# B&R Automation Studio project NAEUL004C00R13L518F00 (part 32)

### Startup.typ - Do Not Change!!!
```iecst
(*2019-04-04*)
(**)

TYPE
	eStartupAction :
		(
		StartupActIdle,
		StartupActRun
		);
	eStartupStep :
		(
		StartupStepUsrFolder,
		StartupStepParameter,
		StartupStepGetHWInfo,
		StartupStepLibVer,
		StartupStepRecipe,
		StartupStepAutoRcp,
		StartupStepUsrMgmt,
		StartupStepBffr,
		StartupStepAlarm,
		StartupStepHermes,
		StartupStepSDOWrite,
		StartupStepSetupUI,
		StartupStepDone
		);
	tyStartUp : 	STRUCT
		In : tyStartUpIn1;
		Out : tyStartUpOut1;
	END_STRUCT;
	tyStartUpOut1 : 	STRUCT
		bRun : BOOL;
		eUsrFolderAct : eUsrFolderAction;
		eHWInfoAct : eHWInfoAction;
		eLibVerAct : eLibVerAction;
		eNtParamAct : eNtParamAction;
		eMcParamAct : eMcParamAction;
		eProdRcpAct : eProdRcpAction;
		eMpProdRcpAct : eMpProdRcpAction;
		eMagRcpAct : eMagRcpAction;
		eUsrMgmtAct : eUsrMgmtAction;
		eBuffer1Act : eBufferAction;
		eBuffer2Act : eBufferAction;
		eBuffer3Act : eBufferAction;
		eAlarmAct : eAlarmAction;
		eUIAct : eUIAction;
		eAWPushPulAct : eAWAction;
		eAWAct : eAWAction;
		eTravAct : eTravAction;
		eLifterAct : eLifterAction;
		eLifter2Act : eLifterAction;
		eMagAW1Act : eMagAWAction;
		eMagAW2Act : eMagAWAction;
		eMagAW3Act : eMagAWAction;
		eHermesAct : eHermesAction;
		eRmtHermesAct : eHermesAction;
		eSvyHermesAct : eHermesAction;
		eAutoRcpAct : eAutoRcpAction;
		eUSHermesAAct : eHermesAction;
		eUSHermesBAct : eHermesAction;
		eServoPPActs : ePullerPusherAction;
		eStartupStep1 : eStartupStep;
		bNtSettingsLoadDone : BOOL := FALSE;
		bUISettingsLoadDone : BOOL;
		sStepTxt : STRING[80];
		bGetConfigDone : BOOL;
		bMismatchSetConfigDone : BOOL;
		eStat : eStartupAction := StartupActIdle;
		eStatus : eFBStatus := Idle;
		sStatTxt : STRING[200] := '';
	END_STRUCT;
	tyStartUpIn1 : 	STRUCT
		eAct : eStartupAction;
	END_STRUCT;
END_TYPE
```

### Startup.var - Change By Project
```iecst
(*2019-05-04*)
VAR
	g_tyStartUp : tyStartUpOut1;
END_VAR
(**)
(*Action & State & Status*)
VAR
	p_StartupStat : UDINT;
	p_StartupStatus : UDINT;
	p_StartupStatTxt : UDINT;
END_VAR
(**)
(*Alarm*)
(**)
(*Output*)
VAR
	p_StartupRun : UDINT;
	p_StartupUsrFolderAct : UDINT;
	p_StartupHWInfoAct : UDINT;
	p_StartupLibVerAct : UDINT;
	p_StartupNtParamAct : UDINT;
	p_StartupMcParamAct : UDINT;
	p_StartupProdRcpAct : UDINT;
	p_StartupMpProdRcpAct : UDINT;
	p_StartupMagRcpAct : UDINT;
	p_StartupUsrMgmtAct : UDINT;
	p_StartupBuffer1Act : UDINT;
	p_StartupBuffer2Act : UDINT;
	p_StartupBuffer3Act : UDINT;
	p_StartupAlarmAct : UDINT;
	p_StartupUIAct : UDINT;
	p_StartupAWAct : UDINT;
	p_StartupAWPushPulAct : UDINT;
	p_StartupTravAct : UDINT;
	p_StartupLifterAct : UDINT;
	p_StartupLifter2Act : {REDUND_UNREPLICABLE} UDINT;
	p_StartupMagAW1Act : UDINT;
	p_StartupMagAW2Act : UDINT;
	p_StartupMagAW3Act : UDINT;
	p_StartupHermesAct : UDINT;
	p_StartupRmtHermesAct : UDINT;
	p_StartupUSHermesAAct : UDINT;
	p_StartupUSHermesBAct : UDINT;
	p_StartupStep : UDINT;
	p_StartupNtSettingsLoadDone : UDINT;
	p_StartupUISettingsLoadDone : UDINT;
	p_StartupStepTxt : UDINT;
	p_StartupGetConfigDone : UDINT;
	p_StartupMismatchSetConfigDone : UDINT;
	p_StartupServoPPAct : UDINT;
	p_StartupSvyHermesAct : UDINT;
	p_StartupAutoRcpsAct : UDINT;
END_VAR
```

### Program Logical/Startup/Startup (IEC, version 1.00.0) - 1.00.0 - 

#### Act_InputConfig.st - Change By Project
```iecst
ACTION Act_InputConfig:

     tylocalStartup.In.eAct := g_tyUIOut.eMnlAct.eStartupAct;

END_ACTION
```

#### Act_OutputConfig.st - Change By Project
```iecst
ACTION Act_OutputConfig:

	g_tyStartUp := tylocalStartup.Out;

	p_StartupProdRcpAct 	:= ADR(tylocalStartup.Out.eProdRcpAct);
	p_StartupMpProdRcpAct 	:= ADR(tylocalStartup.Out.eMpProdRcpAct);

END_ACTION
```

#### Cyclic.st - Do Not Change!!!
```iecst
PROGRAM _CYCLIC

	Act_InputConfig;
	Act_Main;
	Act_OutputConfig;

END_PROGRAM
```

#### Act_Main.st - Change By Project
```iecst
(** 2019-03-28 **)
ACTION Act_Main:
		//Reset Done
	IF tylocalStartup.Out.eStatus = Done AND tylocalStartup.In.eAct = StartupActIdle THEN
		tylocalStartup.Out.eStat	:= StartupActIdle;
	END_IF

	//Set p_eAct
	IF tylocalStartup.Out.eStatus = Idle THEN
		tylocalStartup.Out.eStat	:= tylocalStartup.In.eAct;
	END_IF
	//Main
	CASE tylocalStartup.Out.eStat OF

		StartupActIdle:
			IF tylocalStartup.Out.eStatus <> Idle THEN	//Reset Data
				//Private
				tylocalStartup.Out.eStartupStep1	:= StartupStepUsrFolder;
				tylocalStartup.Out.bRun			:= FALSE;
				usiStep			:= 0;

				tylocalStartup.Out.sStatTxt	:= a_sStatText[tylocalStartup.Out.eStat];

			END_IF

			tylocalStartup.Out.eStatus	:= Idle;

		StartupActRun:
			IF tylocalStartup.Out.eStatus = Idle OR tylocalStartup.Out.eStatus = Busy THEN

				tylocalStartup.Out.eStatus	:= Busy;

				tylocalStartup.Out.sStatTxt	:= a_sStatText[tylocalStartup.Out.eStat];

				tylocalStartup.Out.bRun	:= TRUE;

				CASE tylocalStartup.Out.eStartupStep1 OF

					StartupStepUsrFolder:
						Act_Main_UsrFolder;

					StartupStepParameter:
						Act_Main_Parameter;

					StartupStepGetHWInfo:
						Act_Main_GetHWInfo;

					StartupStepLibVer:
						Act_Main_LibVer;

					StartupStepRecipe:
						Act_Main_Recipe;

					StartupStepAutoRcp:
						IF g_tyNtParamCurr.bAutoRcpPrep AND NOT(g_tyMcParamCurr.bAutoRcpDisable) THEN
							Act_Main_AutoRcp;

						ELSE
							tylocalStartup.Out.eStartupStep1:= StartupStepUsrMgmt;
						END_IF
					StartupStepUsrMgmt:
						Act_Main_UsrMgmt;

					StartupStepBffr:
						Act_Main_Bffr;

					StartupStepAlarm:
						Act_Main_Alarm;

					StartupStepHermes:
						Act_Main_Hermes;

					StartupStepSDOWrite:
						IF DiagCpuIsSimulated() = FALSE THEN
							Act_Main_SDOWrite;
						ELSE
							tylocalStartup.Out.eStartupStep1	:= StartupStepSetupUI;
						END_IF

					StartupStepSetupUI:
						Act_Main_SetupUI;

					StartupStepDone:
						Act_Main_Done;

				END_CASE

				tylocalStartup.Out.sStepTxt	:= a_sStepText[tylocalStartup.Out.eStartupStep1];

			END_IF

	END_CASE

END_ACTION
```

#### Package Logical/Startup/Startup/Act_Main - Change By Project

#### Act_Main_UsrFolder.st
```iecst
(** 2019-05-09 **)
ACTION Act_Main_UsrFolder:

	CASE usiStep OF
		0:
			tylocalStartup.Out.eUsrFolderAct	:= UsrFolderActCreateUsrDir;

			IF (g_tyUsrFolder.eStatus = Done) AND (g_tyUsrFolder.eStat = UsrFolderActCreateUsrDir) THEN

				tylocalStartup.Out.eUsrFolderAct	:= UsrFolderActIdle;
				usiStep			:= 1;

			ELSIF g_tyUsrFolder.eStatus = Error THEN

				tylocalStartup.Out.eUsrFolderAct	:= UsrFolderActIdle;
				tylocalStartup.Out.eStartupStep1	:= StartupStepParameter;

			END_IF

		1:
			tylocalStartup.Out.eUsrFolderAct	:= UsrFolderActCreatePrivateDir;

			IF (g_tyUsrFolder.eStatus = Done) AND (g_tyUsrFolder.eStat = UsrFolderActCreatePrivateDir) THEN

				tylocalStartup.Out.eUsrFolderAct	:= UsrFolderActIdle;
				usiStep			:= 2;

			ELSIF g_tyUsrFolder.eStatus = Error THEN

				tylocalStartup.Out.eUsrFolderAct	:= UsrFolderActIdle;
				usiStep			:= 0;
				tylocalStartup.Out.eStartupStep1	:= StartupStepParameter;

			END_IF

		2:
			tylocalStartup.Out.eUsrFolderAct	:= UsrFolderActCreateLogDir;

			IF (g_tyUsrFolder.eStatus = Done) AND (g_tyUsrFolder.eStat = UsrFolderActCreateLogDir) THEN

				tylocalStartup.Out.eUsrFolderAct	:= UsrFolderActIdle;
				usiStep			:= 3;

			ELSIF g_tyUsrFolder.eStatus = Error THEN

				tylocalStartup.Out.eUsrFolderAct	:= UsrFolderActIdle;
				usiStep			:= 0;
				tylocalStartup.Out.eStartupStep1	:= StartupStepParameter;

			END_IF

		3:
			tylocalStartup.Out.eUsrFolderAct	:= UsrFolderActCreateLCSDir;

			IF (g_tyUsrFolder.eStatus = Done) AND (g_tyUsrFolder.eStat = UsrFolderActCreateLCSDir) THEN

				tylocalStartup.Out.eUsrFolderAct	:= UsrFolderActIdle;
				usiStep			:= 0;
				tylocalStartup.Out.eStartupStep1	:= StartupStepParameter;

			ELSIF g_tyUsrFolder.eStatus = Error THEN

				tylocalStartup.Out.eUsrFolderAct	:= UsrFolderActIdle;
				usiStep			:= 0;
				tylocalStartup.Out.eStartupStep1	:= StartupStepParameter;

			END_IF

	END_CASE

END_ACTION
```

#### Act_Main_GetHWInfo.st
```iecst
(** 2020-10-05 **)
ACTION Act_Main_GetHWInfo:

	CASE usiStep OF
		0:
			tylocalStartup.Out.eHWInfoAct	:= HWInfoActGetIPAddr;

			IF (g_tyHWInfo.eStatus = Done) AND (g_tyHWInfo.eStat = HWInfoActGetIPAddr) THEN

				tylocalStartup.Out.eHWInfoAct		:= HWInfoActIdle;
				usiStep			:= 1;

			ELSIF g_tyHWInfo.eStatus = Error THEN

				tylocalStartup.Out.eHWInfoAct		:= HWInfoActIdle;
				tylocalStartup.Out.eStartupStep1	:= StartupStepLibVer;

			END_IF

		1:
			tylocalStartup.Out.eHWInfoAct	:= HWInfoActGetMacAddr;

			IF (g_tyHWInfo.eStatus = Done) AND (g_tyHWInfo.eStat = HWInfoActGetMacAddr) THEN

				tylocalStartup.Out.eHWInfoAct		:= HWInfoActIdle;
				usiStep			:= 2;

			ELSIF g_tyHWInfo.eStatus = Error THEN

				tylocalStartup.Out.eHWInfoAct		:= HWInfoActIdle;
				usiStep			:= 0;
				tylocalStartup.Out.eStartupStep1	:= StartupStepLibVer;

			END_IF

		2:
			tylocalStartup.Out.eHWInfoAct	:= HWInfoActGetSubnetMask;

			IF (g_tyHWInfo.eStatus = Done) AND (g_tyHWInfo.eStat = HWInfoActGetSubnetMask) THEN

				tylocalStartup.Out.eHWInfoAct		:= HWInfoActIdle;

				IF DiagCpuIsSimulated() = TRUE THEN
					usiStep			:= 0;
					tylocalStartup.Out.eStartupStep1	:= StartupStepLibVer;
				ELSE
					usiStep			:= 3;
				END_IF

			ELSIF g_tyHWInfo.eStatus = Error THEN

				tylocalStartup.Out.eHWInfoAct		:= HWInfoActIdle;
				usiStep			:= 0;
				tylocalStartup.Out.eStartupStep1	:= StartupStepLibVer;

			END_IF

		3:
			tylocalStartup.Out.eHWInfoAct	:= HWInfoActGetEthConfigMode;

			IF (g_tyHWInfo.eStatus = Done) AND (g_tyHWInfo.eStat = HWInfoActGetEthConfigMode) THEN

				tylocalStartup.Out.eHWInfoAct		:= HWInfoActIdle;

				bGetConfigDone	:= TRUE;

				IF (p_tyMcParamCurr.eNetworkMod = UDINT_TO_DINT(p_udiHWInfoEthMode))  THEN
					IF p_udiHWInfoEthMode = DINT_TO_UDINT(IPFromDHCPServer) THEN
						usiStep			:= 0;
						tylocalStartup.Out.eStartupStep1	:= StartupStepLibVer;
					ELSE
						IF (p_tyMcParamCurr.sIPAddr <> p_sHWInfoIPAddr) OR (p_tyMcParamCurr.sSubnetMask <> p_sHWInfoSubnetMask) THEN
							IF g_tyUIOut.bIPTempAddrFillDone AND g_tyUIOut.bIPMismatchOverWriteConfig THEN
								IF (p_tyMcParamCurr.sIPAddr <> p_sHWInfoIPAddr) THEN
									usiStep			:= 5;  //mismatch ip
								ELSE
									usiStep			:= 6;  //mismatch subnet
								END_IF
							END_IF
						ELSE
							usiStep			:= 0;
							tylocalStartup.Out.eStartupStep1	:= StartupStepLibVer;
						END_IF
					END_IF

				ELSE
					IF g_tyUIOut.bIPTempAddrFillDone AND g_tyUIOut.bIPMismatchOverWriteConfig THEN
						usiStep			:= 4;
					END_IF
				END_IF

			ELSIF g_tyHWInfo.eStatus = Error THEN

				tylocalStartup.Out.eHWInfoAct		:= HWInfoActIdle;
				usiStep			:= 0;
				tylocalStartup.Out.eStartupStep1	:= StartupStepLibVer;

			END_IF

		4:
			tylocalStartup.Out.eHWInfoAct	:= HWInfoActSetEthConfigMode;

			IF (g_tyHWInfo.eStatus = Done) AND (g_tyHWInfo.eStat = HWInfoActSetEthConfigMode) THEN

				tylocalStartup.Out.eHWInfoAct		:= HWInfoActIdle;

				IF (p_tyMcParamCurr.eNetworkMod = IPFromDHCPServer) THEN
					usiStep			:= 7;
					bMismatchSetConfigDone	:= TRUE;
				ELSE
					usiStep			:= 5;
				END_IF

			ELSIF g_tyHWInfo.eStatus = Error THEN

				tylocalStartup.Out.eHWInfoAct		:= HWInfoActIdle;
				usiStep			:= 0;
				tylocalStartup.Out.eStartupStep1	:= StartupStepLibVer;

			END_IF

		5:
			tylocalStartup.Out.eHWInfoAct	:= HWInfoActSetIPAddr;

			IF (g_tyHWInfo.eStatus = Done) AND (g_tyHWInfo.eStat = HWInfoActSetIPAddr) THEN

				tylocalStartup.Out.eHWInfoAct		:= HWInfoActIdle;

				IF (p_tyMcParamCurr.sSubnetMask <> p_sHWInfoSubnetMask) THEN
					usiStep			:= 6;
				ELSE
					usiStep			:= 7;
					bMismatchSetConfigDone	:= TRUE;
				END_IF

			ELSIF g_tyHWInfo.eStatus = Error THEN

				tylocalStartup.Out.eHWInfoAct		:= HWInfoActIdle;
				usiStep			:= 0;
				tylocalStartup.Out.eStartupStep1	:= StartupStepLibVer;

			END_IF

		6:
			tylocalStartup.Out.eHWInfoAct	:= HWInfoActSetSubnetMask;

			IF (g_tyHWInfo.eStatus = Done) AND (g_tyHWInfo.eStat = HWInfoActSetSubnetMask) THEN

				tylocalStartup.Out.eHWInfoAct		:= HWInfoActIdle;
				usiStep			:= 7;

				bMismatchSetConfigDone	:= TRUE;

			ELSIF g_tyHWInfo.eStatus = Error THEN

				tylocalStartup.Out.eHWInfoAct		:= HWInfoActIdle;
				usiStep			:= 0;
				tylocalStartup.Out.eStartupStep1	:= StartupStepLibVer;

			END_IF

		7:
			IF g_tyUIOut.bIPConfigChgDone THEN
				IF g_tyUIOut.bOverwriteEthMode THEN
					usiStep			:= 8; //Overwrite Network Mode
				ELSIF g_tyUIOut.bOverwriteIP THEN
					usiStep			:= 9; //Overwrite IP
				ELSIF g_tyUIOut.bOverwriteSubnet THEN
					usiStep			:= 10; //Overwrite Subnet
				ELSE
					usiStep			:= 12; //Load Machine Setting
				END_IF
			END_IF

		8:
			tylocalStartup.Out.eHWInfoAct	:= HWInfoActSetEthConfigMode;

			IF (g_tyHWInfo.eStatus = Done) AND (g_tyHWInfo.eStat = HWInfoActSetEthConfigMode) THEN

				tylocalStartup.Out.eHWInfoAct		:= HWInfoActIdle;

				IF g_tyUIOut.bOverwriteIP THEN
					usiStep			:= 9;
				ELSIF g_tyUIOut.bOverwriteSubnet THEN
					usiStep			:= 10;
				ELSE
					usiStep			:= 11;
				END_IF

			ELSIF g_tyHWInfo.eStatus = Error THEN

				tylocalStartup.Out.eHWInfoAct		:= HWInfoActIdle;
				usiStep			:= 0;
				tylocalStartup.Out.eStartupStep1	:= StartupStepLibVer;

			END_IF

		9:
			tylocalStartup.Out.eHWInfoAct	:= HWInfoActSetIPAddr;

			IF (g_tyHWInfo.eStatus = Done) AND (g_tyHWInfo.eStat = HWInfoActSetIPAddr) THEN

				tylocalStartup.Out.eHWInfoAct		:= HWInfoActIdle;

				IF g_tyUIOut.bOverwriteSubnet THEN
					usiStep			:= 10;
				ELSE
					usiStep			:= 11;
				END_IF

			ELSIF g_tyHWInfo.eStatus = Error THEN

				tylocalStartup.Out.eHWInfoAct		:= HWInfoActIdle;
				usiStep			:= 0;
				tylocalStartup.Out.eStartupStep1	:= StartupStepLibVer;

			END_IF

		10:
			tylocalStartup.Out.eHWInfoAct	:= HWInfoActSetSubnetMask;

			IF (g_tyHWInfo.eStatus = Done) AND (g_tyHWInfo.eStat = HWInfoActSetSubnetMask) THEN

				tylocalStartup.Out.eHWInfoAct		:= HWInfoActIdle;
				usiStep			:= 11;

			ELSIF g_tyHWInfo.eStatus = Error THEN

				tylocalStartup.Out.eHWInfoAct		:= HWInfoActIdle;
				usiStep			:= 0;
				tylocalStartup.Out.eStartupStep1	:= StartupStepLibVer;

			END_IF

		11:

			eMcParamAct	:= McParamActWrite;

			IF (p_eMcParamStatus = Done) AND (p_eMcParamStat = McParamActWrite) THEN

				eMcParamAct		:= McParamActIdle;

				usiStep			:= 12;

			ELSIF p_eMcParamStatus = Error THEN

				eMcParamAct		:= McParamActIdle;
				usiStep			:= 0;
				tylocalStartup.Out.eStartupStep1	:= StartupStepLibVer;

			END_IF

		12:
			tylocalStartup.Out.eHWInfoAct	:= HWInfoActGetIPAddr;

			IF (g_tyHWInfo.eStatus = Done) AND (g_tyHWInfo.eStat = HWInfoActGetIPAddr) THEN

				tylocalStartup.Out.eHWInfoAct		:= HWInfoActIdle;
				usiStep			:= 13;

			ELSIF g_tyHWInfo.eStatus = Error THEN

				tylocalStartup.Out.eHWInfoAct		:= HWInfoActIdle;
				usiStep			:= 0;
				tylocalStartup.Out.eStartupStep1	:= StartupStepLibVer;

			END_IF

		13:
			tylocalStartup.Out.eHWInfoAct	:= HWInfoActGetSubnetMask;

			IF (g_tyHWInfo.eStatus = Done) AND (g_tyHWInfo.eStat = HWInfoActGetSubnetMask) THEN

				tylocalStartup.Out.eHWInfoAct		:= HWInfoActIdle;
				usiStep			:= 0;
				tylocalStartup.Out.eStartupStep1	:= StartupStepLibVer;

			ELSIF g_tyHWInfo.eStatus = Error THEN

				tylocalStartup.Out.eHWInfoAct		:= HWInfoActIdle;
				usiStep			:= 0;
				tylocalStartup.Out.eStartupStep1	:= StartupStepLibVer;

			END_IF

	END_CASE

END_ACTION
```

#### Act_Main_LibVer.st
```iecst
(** 2019-03-28 **)
ACTION Act_Main_LibVer:

	CASE usiStep OF
		0:
			eLibVerAct	:= LibVerActCreateDir;

			IF (p_eLibVerStatus = Done) AND (p_eLibVerStat = LibVerActCreateDir) THEN

				eLibVerAct		:= LibVerActIdle;
				usiStep			:= 1;

			ELSIF p_eLibVerStatus = Error THEN

				eLibVerAct		:= LibVerActIdle;
				tylocalStartup.Out.eStartupStep1	:= StartupStepRecipe;

			END_IF

		1:
			eLibVerAct	:= LibVerActReadChk;

			IF (p_eLibVerStatus = Done) AND (p_eLibVerStat = LibVerActReadChk) THEN

				eLibVerAct		:= LibVerActIdle;
				usiStep			:= 0;
				tylocalStartup.Out.eStartupStep1	:= StartupStepRecipe;

			ELSIF p_eLibVerStatus = Error THEN

				eLibVerAct		:= LibVerActIdle;
				usiStep			:= 0;
				tylocalStartup.Out.eStartupStep1	:= StartupStepRecipe;

			END_IF

	END_CASE

END_ACTION
```

#### Act_Main_Parameter.st
```iecst
(** 2019-03-28 **)
ACTION Act_Main_Parameter:

	CASE usiStep OF
		0:
			tylocalStartup.Out.eNtParamAct	:= NtParamActCreateDir;

			IF (g_tyNtParamOut.eStatus = Done) AND (g_tyNtParamOut.eStat = NtParamActCreateDir) THEN

				tylocalStartup.Out.eNtParamAct			:= NtParamActIdle;
				usiStep				:= 1;

			ELSIF g_tyNtParamOut.eStatus = Error THEN

				bNtSettingsLoadDone	:= TRUE;
				tylocalStartup.Out.eNtParamAct			:= NtParamActIdle;
				usiStep				:= 2;

			END_IF

		1:
			tylocalStartup.Out.eNtParamAct	:= NtParamActRead;

			IF (g_tyNtParamOut.eStatus = Done) AND (g_tyNtParamOut.eStat = NtParamActRead) THEN

				bNtSettingsLoadDone	:= TRUE;
				tylocalStartup.Out.eNtParamAct			:= NtParamActIdle;
				usiStep				:= 2;

			ELSIF g_tyNtParamOut.eStatus = Error THEN

				bNtSettingsLoadDone	:= TRUE;
				tylocalStartup.Out.eNtParamAct			:= NtParamActIdle;
				usiStep				:= 2;

			END_IF

		2:
			tylocalStartup.Out.eMcParamAct	:= McParamActCreateDir;

			IF (g_tyMcParamOut.eStatus = Done) AND (g_tyMcParamOut.eStat = McParamActCreateDir) THEN

				tylocalStartup.Out.eMcParamAct		:= McParamActIdle;
				usiStep			:= 3;

			ELSIF g_tyMcParamOut.eStatus = Error THEN

				tylocalStartup.Out.eMcParamAct		:= McParamActIdle;
				usiStep			:= 0;
				tylocalStartup.Out.eStartupStep1	:= StartupStepGetHWInfo;

			END_IF

		3:
			tylocalStartup.Out.eMcParamAct	:= McParamActRead;

			IF (g_tyMcParamOut.eStatus = Done) AND (g_tyMcParamOut.eStat = McParamActRead) THEN

				tylocalStartup.Out.eMcParamAct		:= McParamActIdle;
				usiStep			:= 0;
				tylocalStartup.Out.eStartupStep1	:= StartupStepGetHWInfo;

			ELSIF g_tyMcParamOut.eStatus = Error THEN

				tylocalStartup.Out.eMcParamAct		:= McParamActIdle;
				usiStep			:= 0;
				tylocalStartup.Out.eStartupStep1	:= StartupStepGetHWInfo;

			END_IF

	END_CASE

END_ACTION
```

#### Act_Main_AutoRcp.st
```iecst
(** 2019-05-04 **)
ACTION Act_Main_AutoRcp:

	CASE usiStep OF
		0:
			tylocalStartup.Out.eAutoRcpAct	:= AutoRcpActCreateDir;

			IF (g_tyAutoRcp.eStatus = Done) AND (g_tyAutoRcp.eStat = AutoRcpActCreateDir) THEN

				tylocalStartup.Out.eAutoRcpAct		:= AutoRcpActIdle;
				usiStep			:= 1;

			ELSIF g_tyAutoRcp.eStatus = Error THEN

				tylocalStartup.Out.eAutoRcpAct		:= AutoRcpActIdle;
				usiStep			:= 1;

			END_IF

		1:
			tylocalStartup.Out.eAutoRcpAct	:= AutoRcpActReadRetain;

			IF (g_tyAutoRcp.eStatus = Done) AND (g_tyAutoRcp.eStat = AutoRcpActReadRetain) THEN
				tylocalStartup.Out.eAutoRcpAct		:= AutoRcpActIdle;
				IF  g_tyNtParamOut.eAutoRcpPrecededBy  = PrecededBySelf THEN
					usiStep			:= 2;
				ELSIF g_tyNtParamOut.eAutoRcpPrecededBy  = PrecededByF1 THEN
					usiStep			:= 0;
					tylocalStartup.Out.eStartupStep1	:= StartupStepUsrMgmt;
				END_IF
			ELSIF g_tyAutoRcp.eStatus = Error THEN
					tylocalStartup.Out.eAutoRcpAct		:= AutoRcpActIdle;
				IF  g_tyNtParamOut.eAutoRcpPrecededBy  = PrecededBySelf THEN
					usiStep			:= 2;
				ELSIF g_tyNtParamOut.eAutoRcpPrecededBy  = PrecededByF1 THEN
					usiStep			:= 0;
					tylocalStartup.Out.eStartupStep1	:= StartupStepUsrMgmt;
				END_IF
			END_IF

		2:
			tylocalStartup.Out.eAutoRcpAct	:= AutoRcpActReadRetain2;

			IF (g_tyAutoRcp.eStatus = Done) AND (g_tyAutoRcp.eStat = AutoRcpActReadRetain2) THEN

				tylocalStartup.Out.eAutoRcpAct		:= AutoRcpActIdle;
				usiStep			:= 0;
				tylocalStartup.Out.eStartupStep1	:= StartupStepUsrMgmt;

			ELSIF g_tyAutoRcp.eStatus = Error THEN

				tylocalStartup.Out.eAutoRcpAct		:= AutoRcpActIdle;
				usiStep			:= 0;
				tylocalStartup.Out.eStartupStep1	:= StartupStepUsrMgmt;

			END_IF

	END_CASE

END_ACTION
```

#### Act_Main_Recipe.st
```iecst
(** 2019-05-04 **)
ACTION Act_Main_Recipe:

	CASE usiStep OF
		0:
			tylocalStartup.Out.eProdRcpAct	:= ProdRcpActCreateDir;

			IF (g_tyProdRcp.eStatus = Done) AND (g_tyProdRcp.eStat = ProdRcpActCreateDir) THEN

				tylocalStartup.Out.eProdRcpAct		:= ProdRcpActIdle;
				usiStep			:= 1;

			ELSIF g_tyProdRcp.eStatus = Error THEN

				tylocalStartup.Out.eProdRcpAct		:= ProdRcpActIdle;
				usiStep			:= 10;

			END_IF

		1:
			tylocalStartup.Out.eProdRcpAct	:= ProdRcpActGetList;

			IF (g_tyProdRcp.eStatus = Done) AND (g_tyProdRcp.eStat = ProdRcpActGetList) THEN

				tylocalStartup.Out.eProdRcpAct		:= ProdRcpActIdle;
				usiStep			:= 2;

			ELSIF g_tyProdRcp.eStatus = Error THEN

				tylocalStartup.Out.eProdRcpAct		:= ProdRcpActIdle;
				usiStep			:= 10;

			END_IF

		2:
			tylocalStartup.Out.eProdRcpAct	:= ProdRcpActReadCurrRcp;

			IF (g_tyProdRcp.eStatus = Done) AND (g_tyProdRcp.eStat = ProdRcpActReadCurrRcp) THEN

				tylocalStartup.Out.eProdRcpAct		:= ProdRcpActIdle;
				usiStep			:= 10;

			ELSIF g_tyMpProdRcp.eStatus = Error THEN

				tylocalStartup.Out.eProdRcpAct		:= ProdRcpActIdle;
				usiStep			:= 10;

			END_IF

		10:
			tylocalStartup.Out.eMpProdRcpAct	:= MpProdRcpActCreateDir;

			IF (g_tyMpProdRcp.eStatus = Done) AND (g_tyMpProdRcp.eStat = MpProdRcpActCreateDir) THEN

				tylocalStartup.Out.eMpProdRcpAct	:= MpProdRcpActIdle;
				usiStep			:= 20;

			ELSIF g_tyMpProdRcp.eStatus = Error THEN

				tylocalStartup.Out.eMpProdRcpAct	:= MpProdRcpActIdle;
				usiStep			:= 20;

			END_IF

		20:
			tylocalStartup.Out.eMagRcpAct	:= MagRcpActCreateDir;

			IF (g_tyMagRcp.eStatus = Done) AND (g_tyMagRcp.eStat = MagRcpActCreateDir) THEN

				tylocalStartup.Out.eMagRcpAct		:= MagRcpActIdle;
				usiStep			:= 21;

			ELSIF g_tyMagRcp.eStatus = Error THEN

				tylocalStartup.Out.eMagRcpAct		:= MagRcpActIdle;
				usiStep			:= 0;
				tylocalStartup.Out.eStartupStep1	:= StartupStepAutoRcp; //StartupStepUsrMgmt;

			END_IF

		21:
			tylocalStartup.Out.eMagRcpAct	:= MagRcpActGetList;

			IF (g_tyMagRcp.eStatus = Done) AND (g_tyMagRcp.eStat = MagRcpActGetList) THEN

				tylocalStartup.Out.eMagRcpAct		:= MagRcpActIdle;
				usiStep			:= 22;

			ELSIF g_tyMagRcp.eStatus = Error THEN

				tylocalStartup.Out.eMagRcpAct		:= MagRcpActIdle;
				usiStep			:= 0;
				tylocalStartup.Out.eStartupStep1	:= StartupStepAutoRcp;

			END_IF

		22:
			tylocalStartup.Out.eMagRcpAct	:= MagRcpActReadCurrRcp;

			IF (g_tyMagRcp.eStatus = Done) AND (g_tyMagRcp.eStat = MagRcpActReadCurrRcp) THEN

				tylocalStartup.Out.eMagRcpAct		:= MagRcpActIdle;
				usiStep			:= 0;
				tylocalStartup.Out.eStartupStep1	:= StartupStepAutoRcp;

			ELSIF g_tyMagRcp.eStatus = Error THEN

				tylocalStartup.Out.eMagRcpAct		:= MagRcpActIdle;
				usiStep			:= 0;
				tylocalStartup.Out.eStartupStep1	:= StartupStepAutoRcp;

			END_IF

	END_CASE

END_ACTION
```

#### Act_Main_UsrMgmt.st
```iecst
(** 2019-03-28 **)
ACTION Act_Main_UsrMgmt:

	CASE usiStep OF
		0:
			tylocalStartup.Out.eUsrMgmtAct	:= UsrMgmtActCreateDir;

			IF (g_tyUsrMgmt.eStatus = Done) AND (g_tyUsrMgmt.eStat = UsrMgmtActCreateDir) THEN

				tylocalStartup.Out.eUsrMgmtAct		:= UsrMgmtActIdle;
				usiStep			:= 1;

			ELSIF g_tyUsrMgmt.eStatus = Error THEN

				tylocalStartup.Out.eUsrMgmtAct		:= UsrMgmtActIdle;
				tylocalStartup.Out.eStartupStep1	:= StartupStepBffr;

			END_IF

		1:
			tylocalStartup.Out.eUsrMgmtAct	:= UsrMgmtActReadData;

			IF (g_tyUsrMgmt.eStatus = Done) AND (g_tyUsrMgmt.eStat = UsrMgmtActReadData) THEN

				tylocalStartup.Out.eUsrMgmtAct		:= UsrMgmtActIdle;
				usiStep			:= 2;

			ELSIF g_tyUsrMgmt.eStatus = Error THEN

				tylocalStartup.Out.eUsrMgmtAct		:= UsrMgmtActIdle;
				usiStep			:= 0;
				tylocalStartup.Out.eStartupStep1	:= StartupStepBffr;

			END_IF

		2:
			tylocalStartup.Out.eUsrMgmtAct	:= UsrMgmtActLogout;

			IF (g_tyUsrMgmt.eStatus = Done) AND (g_tyUsrMgmt.eStat = UsrMgmtActLogout) THEN

				tylocalStartup.Out.eUsrMgmtAct		:= UsrMgmtActIdle;
				usiStep			:= 0;
				tylocalStartup.Out.eStartupStep1	:= StartupStepBffr;

			ELSIF g_tyUsrMgmt.eStatus = Error THEN

				tylocalStartup.Out.eUsrMgmtAct		:= UsrMgmtActIdle;
				usiStep			:= 0;
				tylocalStartup.Out.eStartupStep1	:= StartupStepBffr;

			END_IF

	END_CASE

END_ACTION
```

#### Act_Main_Bffr.st
```iecst
(** 2013-05-27 **)
ACTION Act_Main_Bffr:

	CASE usiStep OF
		//Buffer 1
		0:
			tylocalStartup.Out.eBuffer1Act	:= BufferActCreateDir;

			IF (g_tyBuffer1.eStatus = Done) AND (g_tyBuffer1.eStat = BufferActCreateDir) THEN

				tylocalStartup.Out.eBuffer1Act	:= BufferActIdle;
				usiStep		:= 1;

			ELSIF g_tyBuffer1.eStatus = Error THEN

				tylocalStartup.Out.eBuffer1Act	:= BufferActIdle;
				usiStep		:= 10;

			END_IF

		1:
			tylocalStartup.Out.eBuffer1Act	:= BufferActBGStartBffrSetMty;		//BufferActBGStartBffrSetFull

			IF (g_tyBuffer1.eStatus = Done) AND (g_tyBuffer1.eStat = BufferActBGStartBffrSetMty) THEN		//BufferActBGStartBffrSetFull

				tylocalStartup.Out.eBuffer1Act	:= BufferActIdle;
				usiStep		:= 2;

			ELSIF g_tyBuffer1.eStatus = Error THEN

				tylocalStartup.Out.eBuffer1Act	:= BufferActIdle;
				usiStep		:= 10;

			END_IF

		2:
			IF g_tyBuffer1.bMagPresent = FALSE AND g_tyDI.bMagPresentSen1 = TRUE THEN
				usiStep	:= 4;
			ELSE
				usiStep	:= 3;
			END_IF

		3:
			tylocalStartup.Out.eBuffer1Act	:= BufferActBGStartUpdtSen;

			IF (g_tyBuffer1.eStatus = Done) AND (g_tyBuffer1.eStat = BufferActBGStartUpdtSen) THEN

				tylocalStartup.Out.eBuffer1Act	:= BufferActIdle;
				usiStep		:= 5;

			ELSIF g_tyBuffer1.eStatus = Error THEN

				tylocalStartup.Out.eBuffer1Act	:= BufferActIdle;
				usiStep		:= 10;

			END_IF

		4:
			tylocalStartup.Out.eBuffer1Act	:= BufferActBGStartUpdtSen;

			IF (g_tyBuffer1.eStatus = Done) AND (g_tyBuffer1.eStat = BufferActBGStartUpdtSen) THEN

				tylocalStartup.Out.eBuffer1Act	:= BufferActIdle;
				usiStep		:= 6;

			ELSIF g_tyBuffer1.eStatus = Error THEN

				tylocalStartup.Out.eBuffer1Act	:= BufferActIdle;
				usiStep		:= 10;

			END_IF

		5:
			tylocalStartup.Out.eBuffer1Act	:= BufferActGetRetainBffr;

			IF (g_tyBuffer1.eStatus = Done) AND (g_tyBuffer1.eStat = BufferActGetRetainBffr) THEN

				tylocalStartup.Out.eBuffer1Act	:= BufferActIdle;
				usiStep		:= 7;

			ELSIF g_tyBuffer1.eStatus = Error THEN

				tylocalStartup.Out.eBuffer1Act	:= BufferActIdle;
				usiStep		:= 10;

			END_IF

		6:
			tylocalStartup.Out.eBuffer1Act	:= BufferActSetMty;		//BufferActSetFull

			IF (g_tyBuffer1.eStatus = Done) AND (g_tyBuffer1.eStat = BufferActSetMty) THEN		//BufferActSetFull

				tylocalStartup.Out.eBuffer1Act	:= BufferActIdle;
				usiStep		:= 7;

			ELSIF g_tyBuffer1.eStatus = Error THEN

				tylocalStartup.Out.eBuffer1Act	:= BufferActIdle;
				usiStep		:= 10;

			END_IF

		7:
			tylocalStartup.Out.eBuffer1Act	:= BufferActBGStartCoolFan;

			IF (g_tyBuffer1.eStatus = Done) AND (g_tyBuffer1.eStat = BufferActBGStartCoolFan) THEN

				tylocalStartup.Out.eBuffer1Act		:= BufferActIdle;
				usiStep			:= 10;

			ELSIF g_tyBuffer1.eStatus = Error THEN

				tylocalStartup.Out.eBuffer1Act		:= BufferActIdle;
				usiStep			:= 10;

			END_IF

		//Buffer 2
		10:
			tylocalStartup.Out.eBuffer2Act	:= BufferActCreateDir;

			IF (g_tyBuffer2.eStatus = Done) AND (g_tyBuffer2.eStat = BufferActCreateDir) THEN

				tylocalStartup.Out.eBuffer2Act	:= BufferActIdle;
				usiStep		:= 11;

			ELSIF g_tyBuffer2.eStatus = Error THEN

				tylocalStartup.Out.eBuffer2Act	:= BufferActIdle;
				usiStep		:= 20;

			END_IF

		11:
			tylocalStartup.Out.eBuffer2Act	:= BufferActBGStartBffrSetMty;		//BufferActBGStartBffrSetFull

			IF (g_tyBuffer2.eStatus = Done) AND (g_tyBuffer2.eStat = BufferActBGStartBffrSetMty) THEN		//BufferActBGStartBffrSetFull

				tylocalStartup.Out.eBuffer2Act	:= BufferActIdle;
				usiStep		:= 12;

			ELSIF g_tyBuffer2.eStatus = Error THEN

				tylocalStartup.Out.eBuffer2Act	:= BufferActIdle;
				usiStep		:= 20;

			END_IF

		12:
			IF g_tyBuffer2.bMagPresent = FALSE AND g_tyDI.bMagPresentSen2 = TRUE THEN
				usiStep	:= 14;
			ELSE
				usiStep	:= 13;
			END_IF

		13:
			tylocalStartup.Out.eBuffer2Act	:= BufferActBGStartUpdtSen;

			IF (g_tyBuffer2.eStatus = Done) AND (g_tyBuffer2.eStat = BufferActBGStartUpdtSen) THEN

				tylocalStartup.Out.eBuffer2Act	:= BufferActIdle;
				usiStep		:= 15;

			ELSIF g_tyBuffer2.eStatus = Error THEN

				tylocalStartup.Out.eBuffer2Act	:= BufferActIdle;
				usiStep		:= 20;

			END_IF

		14:
			tylocalStartup.Out.eBuffer2Act	:= BufferActBGStartUpdtSen;

			IF (g_tyBuffer2.eStatus = Done) AND (g_tyBuffer2.eStat = BufferActBGStartUpdtSen) THEN

				tylocalStartup.Out.eBuffer2Act	:= BufferActIdle;
				usiStep		:= 16;

			ELSIF g_tyBuffer2.eStatus = Error THEN

				tylocalStartup.Out.eBuffer2Act	:= BufferActIdle;
				usiStep		:= 20;

			END_IF

		15:
			tylocalStartup.Out.eBuffer2Act	:= BufferActGetRetainBffr;

			IF (g_tyBuffer2.eStatus = Done) AND (g_tyBuffer2.eStat = BufferActGetRetainBffr) THEN

				tylocalStartup.Out.eBuffer2Act	:= BufferActIdle;
				usiStep		:= 17;

			ELSIF g_tyBuffer2.eStatus = Error THEN

				tylocalStartup.Out.eBuffer2Act	:= BufferActIdle;
				usiStep		:= 20;

			END_IF

		16:
			tylocalStartup.Out.eBuffer2Act	:= BufferActSetMty;		//BufferActSetFull

			IF (g_tyBuffer2.eStatus = Done) AND (g_tyBuffer2.eStat = BufferActSetMty) THEN		//BufferActSetFull

				tylocalStartup.Out.eBuffer2Act	:= BufferActIdle;
				usiStep		:= 17;

			ELSIF g_tyBuffer2.eStatus = Error THEN

				tylocalStartup.Out.eBuffer2Act	:= BufferActIdle;
				usiStep		:= 20;

			END_IF

		17:
			tylocalStartup.Out.eBuffer2Act	:= BufferActBGStartCoolFan;

			IF (g_tyBuffer2.eStatus = Done) AND (g_tyBuffer2.eStat = BufferActBGStartCoolFan) THEN

				tylocalStartup.Out.eBuffer2Act		:= BufferActIdle;
				usiStep			:= 20;

			ELSIF g_tyBuffer2.eStatus = Error THEN

				tylocalStartup.Out.eBuffer2Act		:= BufferActIdle;
				usiStep			:= 20;

			END_IF

		//Buffer 3
		20:
			tylocalStartup.Out.eBuffer3Act	:= BufferActCreateDir;

			IF (g_tyBuffer3.eStatus = Done) AND (g_tyBuffer3.eStat = BufferActCreateDir) THEN

				tylocalStartup.Out.eBuffer3Act		:= BufferActIdle;
				usiStep			:= 21;

			ELSIF g_tyBuffer3.eStatus = Error THEN

				tylocalStartup.Out.eBuffer3Act		:= BufferActIdle;
				usiStep			:= 0;
				tylocalStartup.Out.eStartupStep1	:= StartupStepAlarm;

			END_IF

		21:
			tylocalStartup.Out.eBuffer3Act	:= BufferActBGStartBffrSetMty;		//BufferActBGStartBffrSetFull

			IF (g_tyBuffer3.eStatus = Done) AND (g_tyBuffer3.eStat = BufferActBGStartBffrSetMty) THEN		//BufferActBGStartBffrSetFull

				tylocalStartup.Out.eBuffer3Act		:= BufferActIdle;
				usiStep			:= 22;

			ELSIF g_tyBuffer3.eStatus = Error THEN

				tylocalStartup.Out.eBuffer3Act		:= BufferActIdle;
				usiStep			:= 0;
				tylocalStartup.Out.eStartupStep1	:= StartupStepAlarm;

			END_IF

		22:
			IF g_tyBuffer3.bMagPresent = FALSE AND g_tyDI.bMagPresentSen3 = TRUE THEN
				usiStep	:= 24;
			ELSE
				usiStep	:= 23;
			END_IF

		23:
			tylocalStartup.Out.eBuffer3Act	:= BufferActBGStartUpdtSen;

			IF (g_tyBuffer3.eStatus = Done) AND (g_tyBuffer3.eStat = BufferActBGStartUpdtSen) THEN

				tylocalStartup.Out.eBuffer3Act		:= BufferActIdle;
				usiStep			:= 25;

			ELSIF g_tyBuffer3.eStatus = Error THEN

				tylocalStartup.Out.eBuffer3Act		:= BufferActIdle;
				usiStep			:= 0;
				tylocalStartup.Out.eStartupStep1	:= StartupStepAlarm;

			END_IF

		24:
			tylocalStartup.Out.eBuffer3Act	:= BufferActBGStartUpdtSen;

			IF (g_tyBuffer3.eStatus = Done) AND (g_tyBuffer3.eStat = BufferActBGStartUpdtSen) THEN

				tylocalStartup.Out.eBuffer3Act		:= BufferActIdle;
				usiStep			:= 26;

			ELSIF g_tyBuffer3.eStatus = Error THEN

				tylocalStartup.Out.eBuffer3Act		:= BufferActIdle;
				usiStep			:= 0;
				tylocalStartup.Out.eStartupStep1	:= StartupStepAlarm;

			END_IF

		25:
			tylocalStartup.Out.eBuffer3Act	:= BufferActGetRetainBffr;

			IF (g_tyBuffer3.eStatus = Done) AND (g_tyBuffer3.eStat = BufferActGetRetainBffr) THEN

				tylocalStartup.Out.eBuffer3Act		:= BufferActIdle;
				usiStep			:= 27;

			ELSIF g_tyBuffer3.eStatus = Error THEN

				tylocalStartup.Out.eBuffer3Act		:= BufferActIdle;
				usiStep			:= 0;
				tylocalStartup.Out.eStartupStep1	:= StartupStepAlarm;

			END_IF

		26:
			tylocalStartup.Out.eBuffer3Act	:= BufferActSetMty;		//BufferActSetFull

			IF (g_tyBuffer3.eStatus = Done) AND (g_tyBuffer3.eStat = BufferActSetMty) THEN		//BufferActSetFull

				tylocalStartup.Out.eBuffer3Act		:= BufferActIdle;
				usiStep			:= 27;

			ELSIF g_tyBuffer3.eStatus = Error THEN

				tylocalStartup.Out.eBuffer3Act		:= BufferActIdle;
				usiStep			:= 0;
				tylocalStartup.Out.eStartupStep1	:= StartupStepAlarm;

			END_IF

		27:
			tylocalStartup.Out.eBuffer3Act	:= BufferActBGStartCoolFan;

			IF (g_tyBuffer3.eStatus = Done) AND (g_tyBuffer3.eStat = BufferActBGStartCoolFan) THEN

				tylocalStartup.Out.eBuffer3Act		:= BufferActIdle;
				usiStep			:= 0;
				tylocalStartup.Out.eStartupStep1	:= StartupStepAlarm;

			ELSIF g_tyBuffer3.eStatus = Error THEN

				tylocalStartup.Out.eBuffer3Act		:= BufferActIdle;
				usiStep			:= 0;
				tylocalStartup.Out.eStartupStep1	:= StartupStepAlarm;

			END_IF

	END_CASE

END_ACTION
```

#### Act_Main_Alarm.st
```iecst
(** 2019-03-28 **)
ACTION Act_Main_Alarm:

	CASE usiStep OF
		0:
			tylocalStartup.Out.eAlarmAct	:= AlarmActCreateDir;

			IF (g_tyAlm.eStatus = Done) AND (g_tyAlm.eStat = AlarmActCreateDir) THEN

				tylocalStartup.Out.eAlarmAct		:= AlarmActIdle;
				usiStep			:= 1;

			ELSIF g_tyAlm.eStatus = Error THEN

				tylocalStartup.Out.eAlarmAct		:= AlarmActIdle;
				usiStep			:= 0;
				tylocalStartup.Out.eStartupStep1	:= StartupStepHermes;

			END_IF

		1:
			tylocalStartup.Out.eAlarmAct	:= AlarmActDeleteOldLog;

			IF (g_tyAlm.eStatus = Done) AND (g_tyAlm.eStat = AlarmActDeleteOldLog) THEN

				tylocalStartup.Out.eAlarmAct		:= AlarmActIdle;
				usiStep			:= 2;

			ELSIF g_tyAlm.eStatus = Error THEN

				tylocalStartup.Out.eAlarmAct		:= AlarmActIdle;
				usiStep			:= 0;
				tylocalStartup.Out.eStartupStep1	:= StartupStepHermes;

			END_IF

		2:
			tylocalStartup.Out.eAlarmAct	:= AlarmActReadHistory;

			IF (g_tyAlm.eStatus = Done) AND (g_tyAlm.eStat = AlarmActReadHistory) THEN

				tylocalStartup.Out.eAlarmAct		:= AlarmActIdle;
				usiStep			:= 3;

			ELSIF g_tyAlm.eStatus = Error THEN

				tylocalStartup.Out.eAlarmAct		:= AlarmActIdle;
				usiStep			:= 0;
				tylocalStartup.Out.eStartupStep1	:= StartupStepHermes;

			END_IF

		3:
			tylocalStartup.Out.eAlarmAct	:= AlarmActBGStartLog;

			IF (g_tyAlm.eStatus = Done) AND (g_tyAlm.eStat = AlarmActBGStartLog) THEN

				tylocalStartup.Out.eAlarmAct		:= AlarmActIdle;
				usiStep			:= 0;
				tylocalStartup.Out.eStartupStep1	:= StartupStepHermes;

			ELSIF g_tyAlm.eStatus = Error THEN

				tylocalStartup.Out.eAlarmAct		:= AlarmActIdle;
				usiStep			:= 0;
				tylocalStartup.Out.eStartupStep1	:= StartupStepHermes;

			END_IF

	END_CASE

END_ACTION
```

#### Act_Main_Hermes.st
```iecst
(** 2019-05-04 **)
ACTION Act_Main_Hermes:

	CASE usiStep OF
		0:
			tylocalStartup.Out.eHermesAct	:= HermesActCreateDir;

			IF (g_tyHermes.eStatus = Done) AND (g_tyHermes.eStat = HermesActCreateDir) THEN

				tylocalStartup.Out.eHermesAct		:= HermesActIdle;
				usiStep			:= 1;

			ELSIF g_tyHermes.eStatus = Error THEN

				tylocalStartup.Out.eHermesAct		:= HermesActIdle;
				usiStep			:= 10;

			END_IF

		1:
			tylocalStartup.Out.eHermesAct	:= HermesActReadRetainLane1;

			IF (g_tyHermes.eStatus = Done) AND (g_tyHermes.eStat = HermesActReadRetainLane1) THEN

				tylocalStartup.Out.eHermesAct		:= HermesActIdle;
				usiStep			:= 2;

			ELSIF g_tyHermes.eStatus = Error THEN

				tylocalStartup.Out.eHermesAct		:= HermesActIdle;
				usiStep			:= 10;

			END_IF

		2:
			tylocalStartup.Out.eHermesAct	:= HermesActReadConfig;

			IF (g_tyHermes.eStatus = Done) AND (g_tyHermes.eStat = HermesActReadConfig) THEN

				tylocalStartup.Out.eHermesAct		:= HermesActIdle;
				usiStep			:= 10;

			ELSIF g_tyHermes.eStatus = Error THEN

				tylocalStartup.Out.eHermesAct		:= HermesActIdle;
				usiStep			:= 10;

			END_IF

		10:
			tylocalStartup.Out.eUSHermesAAct	:= HermesActDeleteOldLog;

			IF (g_tyUSHermesA.eStatus = Done) AND (g_tyUSHermesA.eStat = HermesActDeleteOldLog) THEN

				tylocalStartup.Out.eUSHermesAAct	:= HermesActIdle;
				usiStep			:= 11;

			ELSIF g_tyUSHermesA.eStatus = Error THEN

				tylocalStartup.Out.eUSHermesAAct	:= HermesActIdle;
				usiStep			:= 11;

			END_IF
		11:
			tylocalStartup.Out.eUSHermesBAct	:= HermesActDeleteOldLog;

			IF (g_tyUSHermesB.eStatus = Done) AND (g_tyUSHermesB.eStat = HermesActDeleteOldLog) THEN

				tylocalStartup.Out.eUSHermesBAct	:= HermesActIdle;
				usiStep			:= 30;

			ELSIF g_tyUSHermesB.eStatus = Error THEN

				tylocalStartup.Out.eUSHermesBAct	:= HermesActIdle;
				usiStep			:= 30;

			END_IF

		30:
			tylocalStartup.Out.eRmtHermesAct	:= HermesActDeleteOldLog;

			IF (g_tyRmtHermes.esStatus = Done) AND (g_tyRmtHermes.esStat = HermesActDeleteOldLog) THEN

				tylocalStartup.Out.eRmtHermesAct	:= HermesActIdle;
				usiStep			:= 40;

//				usiStep			:= 0;  //Changed
//				tylocalStartup.Out.eStartupStep1	:= StartupStepSetupUI; //Changed
			ELSIF g_tyRmtHermes.esStatus = Error THEN

				tylocalStartup.Out.eRmtHermesAct	:= HermesActIdle;
				usiStep			:= 40;

//				usiStep			:= 0;  //Changed
//				tylocalStartup.Out.eStartupStep1	:= StartupStepSetupUI; //Changed
			END_IF

		40:
			tylocalStartup.Out.eSvyHermesAct	:= HermesActDeleteOldLog;

			IF (g_tySvyHermes.eStatus = Done) AND (g_tySvyHermes.eStat = HermesActDeleteOldLog) THEN

				tylocalStartup.Out.eSvyHermesAct	:= HermesActIdle;
				usiStep			:= 42;

			ELSIF g_tySvyHermes.eStatus = Error THEN

				tylocalStartup.Out.eSvyHermesAct	:= HermesActIdle;
				usiStep			:= 42;

			END_IF

		42:
			tylocalStartup.Out.eSvyHermesAct	:= HermesActReadRetainSendWO1;

			IF (g_tySvyHermes.eStatus = Done) AND (g_tySvyHermes.eStat = HermesActReadRetainSendWO1) THEN

				tylocalStartup.Out.eSvyHermesAct	:= HermesActIdle;
				usiStep			:= 43;

			ELSIF g_tySvyHermes.eStatus = Error THEN

				tylocalStartup.Out.eSvyHermesAct	:= HermesActIdle;
				usiStep			:= 43;
			END_IF
		43:
			tylocalStartup.Out.eSvyHermesAct	:= HermesActReadRetainSendWO2;

			IF (g_tySvyHermes.eStatus = Done) AND (g_tySvyHermes.eStat = HermesActReadRetainSendWO2) THEN

				tylocalStartup.Out.eSvyHermesAct	:= HermesActIdle;
				usiStep			:= 44;

			ELSIF g_tySvyHermes.eStatus = Error THEN

				tylocalStartup.Out.eSvyHermesAct	:= HermesActIdle;
				usiStep			:= 44;
			END_IF

		44:
			tylocalStartup.Out.eSvyHermesAct	:= HermesActReadRetainSendWO3;

			IF (g_tySvyHermes.eStatus = Done) AND (g_tySvyHermes.eStat = HermesActReadRetainSendWO3) THEN

				tylocalStartup.Out.eSvyHermesAct	:= HermesActIdle;
				usiStep			:= 0;
				tylocalStartup.Out.eStartupStep1	:= StartupStepSetupUI;
			ELSIF g_tySvyHermes.eStatus = Error THEN

				tylocalStartup.Out.eSvyHermesAct	:= HermesActIdle;

				usiStep			:= 0;
				tylocalStartup.Out.eStartupStep1	:= StartupStepSetupUI;
			END_IF
	END_CASE

END_ACTION
```

#### Act_Main_SDOWrite.st
```iecst
(** 2019-10-21 **)
ACTION Act_Main_SDOWrite:

	CASE usiStep OF

		0:
			tylocalStartup.Out.eAWPushPulAct	:= AWActBGStartModOKChk;

			IF (g_tyAWPushOrPuller.eStatus = Done) AND (g_tyAWPushOrPuller.eStat = AWActBGStartModOKChk) THEN

				tylocalStartup.Out.eAWPushPulAct	:= AWActIdle;
				usiStep		:= 1;

			ELSIF g_tyAWPushOrPuller.eStatus = Error THEN

				tylocalStartup.Out.eAWPushPulAct		:= AWActIdle;
				usiStep		:= 1;

			END_IF

		1:
			tylocalStartup.Out.eAWAct	:= AWActBGStartModOKChk;

			IF (g_tyAW.eStatus = Done) AND (g_tyAW.eStat = AWActBGStartModOKChk) THEN

				tylocalStartup.Out.eAWAct		:= AWActIdle;
		   		usiStep		:= 2;

			ELSIF g_tyAW.eStatus = Error THEN

				tylocalStartup.Out.eAWAct		:= AWActIdle;
				usiStep		:= 2;

			END_IF

		2:
			tylocalStartup.Out.eMagAW1Act	:= MagAWActBGStartModOKChk;

			IF (g_tyMagAW1.eStatus = Done) AND (g_tyMagAW1.eStat = MagAWActBGStartModOKChk) THEN

				tylocalStartup.Out.eMagAW1Act	:= MagAWActIdle;
				usiStep		:= 4;

			ELSIF g_tyMagAW1.eStatus = Error THEN

				tylocalStartup.Out.eMagAW1Act	:= MagAWActIdle;
				usiStep		:= 4;

			END_IF

		4:
			tylocalStartup.Out.eMagAW2Act	:= MagAWActBGStartModOKChk;

			IF (g_tyMagAW2.eStatus = Done) AND (g_tyMagAW2.eStat = MagAWActBGStartModOKChk) THEN

				tylocalStartup.Out.eMagAW2Act	:= MagAWActIdle;
				usiStep		:= 6;

			ELSIF g_tyMagAW2.eStatus = Error THEN

				tylocalStartup.Out.eMagAW2Act	:= MagAWActIdle;
				usiStep		:= 6;

			END_IF

		6:
			tylocalStartup.Out.eMagAW3Act	:= MagAWActBGStartModOKChk;

			IF (g_tyMagAW3.eStatus = Done) AND (g_tyMagAW3.eStat = MagAWActBGStartModOKChk) THEN

				tylocalStartup.Out.eMagAW3Act	:= MagAWActIdle;
				usiStep		:= 10;

			ELSIF g_tyMagAW3.eStatus = Error THEN

				tylocalStartup.Out.eMagAW3Act	:= MagAWActIdle;
				usiStep		:= 10;

			END_IF

		10:
			tylocalStartup.Out.eTravAct	:= TravActBGStartModOKChk;

			IF (g_tyTrav.eStatus = Done) AND (g_tyTrav.eStat = TravActBGStartModOKChk) THEN

				tylocalStartup.Out.eTravAct	:= TravActIdle;
				usiStep		:= 20;

			ELSIF g_tyTrav.eStatus = Error THEN

				tylocalStartup.Out.eTravAct	:= TravActIdle;
				usiStep		:= 20;

			END_IF

		20:
			tylocalStartup.Out.eLifterAct	:= LifterActBGStartModOKChk;

			IF (g_tyLifter.eStatus = Done) AND (g_tyLifter.eStat = LifterActBGStartModOKChk) THEN

				tylocalStartup.Out.eLifterAct		:= LifterActIdle;
				usiStep			:= 21;
				tylocalStartup.Out.eStartupStep1	:= StartupStepSetupUI;

			ELSIF g_tyLifter.eStatus = Error THEN

				tylocalStartup.Out.eLifterAct		:= LifterActIdle;
				usiStep			:= 21;
				tylocalStartup.Out.eStartupStep1	:= StartupStepSetupUI;

			END_IF
		21:
			tylocalStartup.Out.eLifter2Act	:= LifterActBGStartModOKChk;

			IF (g_tyLifter2.eStatus = Done) AND (g_tyLifter2.eStat = LifterActBGStartModOKChk) THEN

				tylocalStartup.Out.eLifter2Act		:= LifterActIdle;
				usiStep			:= 0;
				tylocalStartup.Out.eStartupStep1	:= StartupStepSetupUI;

			ELSIF g_tyLifter2.eStatus = Error THEN

				tylocalStartup.Out.eLifter2Act		:= LifterActIdle;
				usiStep			:= 0;
				tylocalStartup.Out.eStartupStep1	:= StartupStepSetupUI;

			END_IF

	END_CASE

END_ACTION
```

#### Act_Main_SetupUI.st
```iecst
(** 2019-03-28 **)
ACTION Act_Main_SetupUI:

	CASE usiStep OF
		0:
			tylocalStartup.Out.eUIAct	:= UIActInitial;

			IF (g_tyUIOut.eStatus = Done) AND (g_tyUIOut.eStat = UIActInitial) THEN

				tylocalStartup.Out.eUIAct			:= UIActIdle;
				tylocalStartup.Out.eStartupStep1	:= StartupStepDone;
				tylocalStartup.Out.bUISettingsLoadDone := TRUE;
			ELSIF g_tyUIOut.eStatus = Error THEN

				tylocalStartup.Out.eUIAct			:= UIActIdle;
				tylocalStartup.Out.eStartupStep1	:= StartupStepDone;
				tylocalStartup.Out.bUISettingsLoadDone := TRUE;
			END_IF

	END_CASE

END_ACTION
```

#### Local.var - Do Not Change!!!
```iecst
(*2020-09-22*)
VAR
	tylocalStartup : tyStartUp;
END_VAR
(**)
(*Local Action, State & Status*)
VAR
	eAct : eStartupAction := StartupActIdle;
	a_sStatText : ARRAY[0..50] OF STRING[200] := ['Idling','Running Startup',49('')];
END_VAR
(**)
(*All General Alarm*)
VAR
	tyUIAlmData : tyUIAllAlm;
END_VAR
(*Local Alarm*)
(**)
(*Local Output*)
VAR
	a_sStepText : ARRAY[0..12] OF STRING[80] := ['Creating User Folder','Reading Parameter','Getting Hardware Info','Checking Library Version','Reading Recipe List','Reading Retain Magazine Recipe List','Reading User Management List','Reading Buffer / Magazine Data','Setting Up Alarm','Setting Up Hermes','Writing Data To Servo Motor','Setting Up User Interface','Done'];
END_VAR
(**)
(*Local Input*)
VAR
	bMismatchOverWriteConfig : BOOL;
	bTempAddrFillDone : BOOL;
	bChgConfigDone : BOOL;
	bOverwriteIP : BOOL;
	bOverwriteSubnet : BOOL;
	bOverwriteEthMode : BOOL;
	tyNtParamCurr : tyNtParam;
	tyMcParamCurr : tyMcParam;
END_VAR
(**)
(*Local*)
VAR
	bInitDone : BOOL;
	bInitialDone : BOOL;
	usiStep : USINT;
END_VAR
```

#### InputRef_Link.var - not listed in the package file held
```iecst
(*2020-09-22*)
(**)
(*User Folder*)
VAR
	p_eUsrFolderStat : REFERENCE TO eUsrFolderAction;
	p_eUsrFolderStatus : REFERENCE TO eFBStatus;
END_VAR
(**)
(*Hardware Info*)
VAR
	p_eHWInfoStat : REFERENCE TO eHWInfoAction;
	p_eHWInfoStatus : REFERENCE TO eFBStatus;
	p_sHWInfoIPAddr : REFERENCE TO STRING[15];
	p_sHWInfoSubnetMask : REFERENCE TO STRING[15];
	p_udiHWInfoEthMode : REFERENCE TO UDINT;
END_VAR
(**)
(*Library Version*)
VAR
	p_eLibVerStat : REFERENCE TO eLibVerAction;
	p_eLibVerStatus : REFERENCE TO eFBStatus;
END_VAR
(**)
(*Nutek Parameter*)
VAR
	p_eNtParamStat : REFERENCE TO eNtParamAction;
	p_eNtParamStatus : REFERENCE TO eFBStatus;
END_VAR
(**)
(*Machine Parameter*)
VAR
	p_eMcParamStat : REFERENCE TO eMcParamAction;
	p_eMcParamStatus : REFERENCE TO eFBStatus;
END_VAR
(**)
(*Product Recipe*)
VAR
	p_eProdRcpStat : REFERENCE TO eProdRcpAction;
	p_eProdRcpStatus : REFERENCE TO eFBStatus;
END_VAR
(**)
(*Mp Product Recipe*)
VAR
	p_eMpProdRcpStat : REFERENCE TO eMpProdRcpAction;
	p_eMpProdRcpStatus : REFERENCE TO eFBStatus;
END_VAR
(**)
(*Magazine Recipe*)
VAR
	p_eMagRcpStat : REFERENCE TO eMagRcpAction;
	p_eMagRcpStatus : REFERENCE TO eFBStatus;
END_VAR
(**)
(*User Management*)
VAR
	p_eUsrMgmtStat : REFERENCE TO eUsrMgmtAction;
	p_eUsrMgmtStatus : REFERENCE TO eFBStatus;
END_VAR
(**)
(*Buffer*)
VAR
	p_eBuffer1Stat : REFERENCE TO eBufferAction;
	p_eBuffer1Status : REFERENCE TO eFBStatus;
	p_bMagPresentSensor1 : REFERENCE TO BOOL;
	p_bMagPresent1 : REFERENCE TO BOOL;
END_VAR
(**)
VAR
	p_eBuffer2Stat : REFERENCE TO eBufferAction;
	p_eBuffer2Status : REFERENCE TO eFBStatus;
	p_bMagPresentSensor2 : REFERENCE TO BOOL;
	p_bMagPresent2 : REFERENCE TO BOOL;
END_VAR
(**)
VAR
	p_eBuffer3Stat : REFERENCE TO eBufferAction;
	p_eBuffer3Status : REFERENCE TO eFBStatus;
	p_bMagPresentSensor3 : REFERENCE TO BOOL;
	p_bMagPresent3 : REFERENCE TO BOOL;
END_VAR
(**)
(*Alarm Log*)
VAR
	p_eAlarmStat : REFERENCE TO eAlarmAction;
	p_eAlarmStatus : REFERENCE TO eFBStatus;
END_VAR
(**)
(*Hermes*)
VAR
	p_eHermesStat : REFERENCE TO eHermesAction;
	p_eHermesStatus : REFERENCE TO eFBStatus;
END_VAR
(**)
VAR
	p_eRmtHermesStat : REFERENCE TO eHermesAction;
	p_eRmtHermesStatus : REFERENCE TO eFBStatus;
END_VAR
(**)
VAR
	p_eSvyHermesStat : REFERENCE TO eHermesAction;
	p_eSvyHermesStatus : REFERENCE TO eFBStatus;
END_VAR
(**)
VAR
	p_eUSHermesAStat : REFERENCE TO eHermesAction;
	p_eUSHermesAStatus : REFERENCE TO eFBStatus;
END_VAR
(**)
VAR
	p_eUSHermesBStat : REFERENCE TO eHermesAction;
	p_eUSHermesBStatus : REFERENCE TO eFBStatus;
END_VAR
(**)
(*Auto Width*)
VAR
	p_eAWStat : REFERENCE TO eAWAction;
	p_eAWStatus : REFERENCE TO eFBStatus;
END_VAR
(**)
(*Auto Width*)
VAR
	p_eAWPushOrPullerStat : REFERENCE TO eAWAction;
	p_eAWPushOrPullerStatus : REFERENCE TO eFBStatus;
END_VAR
(**)
(*Traverser*)
VAR
	p_eTravStat : REFERENCE TO eTravAction;
	p_eTravStatus : REFERENCE TO eFBStatus;
END_VAR
(**)
(*Lifter*)
VAR
	p_eLifterStat : REFERENCE TO eLifterAction;
	p_eLifterStatus : REFERENCE TO eFBStatus;
	p_eLifter2Stat : REFERENCE TO eLifterAction;
	p_eLifter2Status : REFERENCE TO eFBStatus;
END_VAR
(**)
(*Magazine Auto Width*)
VAR
	p_eMagAW1Stat : REFERENCE TO eMagAWAction;
	p_eMagAW1Status : REFERENCE TO eFBStatus;
END_VAR
(**)
VAR
	p_eMagAW2Stat : REFERENCE TO eMagAWAction;
	p_eMagAW2Status : REFERENCE TO eFBStatus;
END_VAR
(**)
VAR
	p_eMagAW3Stat : REFERENCE TO eMagAWAction;
	p_eMagAW3Status : REFERENCE TO eFBStatus;
END_VAR
(* *)
VAR
	p_bNtParamAutoRcpPrep : REFERENCE TO BOOL;
	p_eNtParamAutoRcpPrecededBy : REFERENCE TO eAutoRcpPreceded;
	p_bMcParamAutoRcpDis : REFERENCE TO BOOL;
	p_eAutoRcpStat : REFERENCE TO eAutoRcpAction;
	p_eAutoRcpStatus : REFERENCE TO eFBStatus;
END_VAR
(**)
(*User Interface*)
VAR
	p_eUIStat : REFERENCE TO eUIAction;
	p_eUIStatus : REFERENCE TO eFBStatus;
END_VAR
```

#### Act_InitGlobal.st - not listed in the package file held
```iecst
(** 2020-09-22 **)
ACTION Act_InitGlobal:

	(* Always Change If Project Change *)

	//Pass Data To Link

	//Pass Data To Internal Use
	p_eAct ACCESS p_UIStartupAct;
	p_tyNtParamCurr ACCESS p_NtParamCurr;
	p_tyMcParamCurr ACCESS p_McParamCurr;

	p_bUIMismatchOverWriteConfig ACCESS p_UIMismatchOverWriteConfig;
	p_bUITempAddrFillDone ACCESS p_UITempAddrFillDone;
	p_bUIChgConfigDone ACCESS p_UIIPConfigChgDone;
	p_bUIOverwriteIP ACCESS p_UIOverwriteIP;
	p_bUIOverwriteSubnet ACCESS p_UIOverwriteSubnet;
	p_bUIOverwriteEthMode ACCESS p_UIOverwriteEthMode;

	p_eUsrFolderStat ACCESS p_UsrFolderStat;
	p_eUsrFolderStatus ACCESS p_UsrFolderStatus;

	p_eHWInfoStat ACCESS p_HWInfoStat;
	p_eHWInfoStatus ACCESS p_HWInfoStatus;
	p_sHWInfoIPAddr ACCESS p_HWInfoIPAddr;
	p_sHWInfoSubnetMask ACCESS p_HWInfoSubnetMask;
	p_udiHWInfoEthMode ACCESS p_HWInfoEthMode;

	p_eLibVerStat ACCESS p_LibVerStat;
	p_eLibVerStatus ACCESS p_LibVerStatus;

	p_eNtParamStat ACCESS p_NtParamStat;
	p_eNtParamStatus ACCESS p_NtParamStatus;

	p_eMcParamStat ACCESS p_McParamStat;
	p_eMcParamStatus ACCESS p_McParamStatus;

	p_eProdRcpStat ACCESS p_ProdRcpStat;
	p_eProdRcpStatus ACCESS p_ProdRcpStatus;

	p_eMpProdRcpStat ACCESS p_MpProdRcpStat;
	p_eMpProdRcpStatus ACCESS p_MpProdRcpStatus;

	p_eMagRcpStat ACCESS p_MagRcpStat;
	p_eMagRcpStatus ACCESS p_MagRcpStatus;

	p_eUsrMgmtStat ACCESS p_UsrMgmtStat;
	p_eUsrMgmtStatus ACCESS p_UsrMgmtStatus;

	p_eBuffer1Stat ACCESS p_Buffer1Stat;
	p_eBuffer1Status ACCESS p_Buffer1Status;
	p_bMagPresentSensor1 ACCESS p_DIMagPresentSen1;
	p_bMagPresent1 ACCESS p_Buffer1MagPresent;

	p_eBuffer2Stat ACCESS p_Buffer2Stat;
	p_eBuffer2Status ACCESS p_Buffer2Status;
	p_bMagPresentSensor2 ACCESS p_DIMagPresentSen2;
	p_bMagPresent2 ACCESS p_Buffer2MagPresent;

	p_eBuffer3Stat ACCESS p_Buffer3Stat;
	p_eBuffer3Status ACCESS p_Buffer3Status;
	p_bMagPresentSensor3 ACCESS p_DIMagPresentSen3;
	p_bMagPresent3 ACCESS p_Buffer3MagPresent;

	p_eAlarmStat ACCESS p_AlarmStat;
	p_eAlarmStatus ACCESS p_AlarmStatus;

	p_eHermesStat ACCESS p_HermesStat;
	p_eHermesStatus ACCESS p_HermesStatus;

	p_eRmtHermesStat ACCESS p_RmtHermesStat;
	p_eRmtHermesStatus ACCESS p_RmtHermesStatus;

	p_eUSHermesAStat ACCESS p_USHermesAStat;
	p_eUSHermesAStatus ACCESS p_USHermesAStatus;

	p_eUSHermesBStat ACCESS p_USHermesBStat;
	p_eUSHermesBStatus ACCESS p_USHermesBStatus;

	p_eSvyHermesStat ACCESS p_SvyHermesStat;//new for Hermes 1.3
	p_eSvyHermesStatus ACCESS p_SvyHermesStatus;//new for Hermes 1.3

	p_eAWPushOrPullerStat ACCESS p_AWPushOrPullerStat;
	p_eAWPushOrPullerStatus ACCESS p_AWPushOrPullerStatus;

	p_eAWStat ACCESS p_AWOpenStat;
	p_eAWStatus ACCESS p_AWOpenStatus;

	p_eTravStat ACCESS p_TravStat;
	p_eTravStatus ACCESS p_TravStatus;

	p_eLifterStat ACCESS p_LifterBtmStat;
	p_eLifterStatus ACCESS p_LifterBtmStatus;

	p_eLifter2Stat ACCESS p_Lifter2Stat;
	p_eLifter2Status ACCESS p_Lifter2Status;

	p_eUIStat ACCESS p_UIStat;
	p_eUIStatus ACCESS p_UIStatus;

	p_eMagAW1Stat ACCESS p_MagAWOpen1Stat;
	p_eMagAW1Status ACCESS p_MagAWOpen1Status;

	p_eMagAW2Stat ACCESS p_MagAWOpen2Stat;
	p_eMagAW2Status ACCESS p_MagAWOpen2Status;

	p_eMagAW3Stat ACCESS p_MagAWOpen3Stat;
	p_eMagAW3Status ACCESS p_MagAWOpen3Status;

	p_bNtParamAutoRcpPrep ACCESS p_NtParamAutoRcpPrep;
	p_eNtParamAutoRcpPrecededBy ACCESS p_NtParamAutoRcpPrecededBy;
	p_bMcParamAutoRcpDis ACCESS p_McParamAutoRcpDisable;
	p_eAutoRcpStat ACCESS p_AutoRcpStat;
	p_eAutoRcpStatus ACCESS p_AutoRcpStatus;

	(* Always Change If Project Change *)

END_ACTION
```

#### Act_InitLocal.st - not listed in the package file held
```iecst
(** 2020-09-22 **)
ACTION Act_InitLocal:

	//Input Reference Link To Local Variable
	p_eAct ACCESS ADR(eAct);
	p_tyNtParamCurr ACCESS ADR(tyNtParamCurr);
	p_tyMcParamCurr ACCESS ADR(tyMcParamCurr);

	p_bUIMismatchOverWriteConfig ACCESS ADR(bMismatchOverWriteConfig);
	p_bUITempAddrFillDone ACCESS ADR(bTempAddrFillDone);
	p_bUIChgConfigDone ACCESS ADR(bChgConfigDone);
	p_bUIOverwriteIP ACCESS ADR(bOverwriteIP);
	p_bUIOverwriteSubnet ACCESS ADR(bOverwriteSubnet);
	p_bUIOverwriteEthMode ACCESS ADR(bOverwriteEthMode);

END_ACTION
```

#### Init.st - not listed in the package file held
```iecst
(** 2019-05-04 **)
PROGRAM _INIT

	(* Always Change If Project Change *)

	//Pass Address To External Use
	p_StartupStat		:= ADR(eStat);
	p_StartupStatus		:= ADR(eStatus);
	p_StartupStatTxt	:= ADR(sStatTxt);

	//Alarm

	//Output
	p_StartupRun				:= ADR(bRun);
	p_StartupUsrFolderAct		:= ADR(eUsrFolderAct);
	p_StartupHWInfoAct			:= ADR(eHWInfoAct);
	p_StartupLibVerAct			:= ADR(eLibVerAct);
	p_StartupNtParamAct			:= ADR(eNtParamAct);
	p_StartupMcParamAct			:= ADR(eMcParamAct);
	p_StartupProdRcpAct			:= ADR(eProdRcpAct);
	p_StartupMpProdRcpAct		:= ADR(eMpProdRcpAct);
	p_StartupMagRcpAct			:= ADR(eMagRcpAct);
	p_StartupUsrMgmtAct			:= ADR(eUsrMgmtAct);
	p_StartupBuffer1Act			:= ADR(eBuffer1Act);
	p_StartupBuffer2Act			:= ADR(eBuffer2Act);
	p_StartupBuffer3Act			:= ADR(eBuffer3Act);
	p_StartupAlarmAct			:= ADR(eAlarmAct);
	p_StartupUIAct				:= ADR(eUIAct);
	p_StartupAWAct				:= ADR(eAWAct);
	p_StartupAWPushPulAct		:= ADR(eAWPushPulAct);
	p_StartupTravAct			:= ADR(eTravAct);
	p_StartupLifterAct			:= ADR(eLifterAct);
	p_StartupLifter2Act			:= ADR(eLifter2Act);
	p_StartupMagAW1Act			:= ADR(eMagAW1Act);
	p_StartupMagAW2Act			:= ADR(eMagAW2Act);
	p_StartupMagAW3Act			:= ADR(eMagAW3Act);
	p_StartupHermesAct			:= ADR(eHermesAct);
	p_StartupRmtHermesAct		:= ADR(eRmtHermesAct);
	p_StartupUSHermesAAct		:= ADR(eUSHermesAAct);
	p_StartupUSHermesBAct		:= ADR(eUSHermesBAct);
	p_StartupStep				:= ADR(eStartupStep1);
	p_StartupNtSettingsLoadDone	:= ADR(bNtSettingsLoadDone);
	p_StartupUISettingsLoadDone := ADR(bUISettingsLoadDone);
	p_StartupStepTxt			:= ADR(sStepTxt);
	p_StartupServoPPAct			:= ADR(eServoPPAct);
	p_StartupSvyHermesAct		:= ADR(eSvyHermesAct); //new for Hermes 1.3
	p_StartupAutoRcpsAct		:= ADR(eAutoRcpAct);

	p_StartupGetConfigDone			:= ADR(bGetConfigDone);
	p_StartupMismatchSetConfigDone	:= ADR(bMismatchSetConfigDone);
	(* Always Change If Project Change *)

END_PROGRAM
```

- Program Logical/General/General (IEC, version 1.00.0) - 1.00.0 - (2018-12-07) (no source held here)

### UsrFolder.typ - Do Not Change!!!
```iecst
(*2019-05-09*)
(**)
(*Action*)

TYPE
	eUsrFolderAction :
		(
		UsrFolderActIdle,
		UsrFolderActCreateUsrDir,
		UsrFolderActCreatePrivateDir,
		UsrFolderActCreateLogDir,
		UsrFolderActCreateLCSDir
		);
	tyUsrFolder : 	STRUCT
		In : tyUsrFolderIn1;
		Out : tyUsrFolderOut1;
	END_STRUCT;
	tyUsrFolderIn1 : 	STRUCT
		eAct : eUsrFolderAction; (*User Folder's Action*)
		udiRstErr : UDINT := 0; (*Reset Error*)
		sProgNm : STRING[15] := 'UsrFolder'; (*Program's Name*)
	END_STRUCT;
	tyUsrFolderOut1 : 	STRUCT
		eStat : eUsrFolderAction := UsrFolderActIdle; (*User Folder's State*)
		eStatus : eFBStatus := Idle; (*User Folder's Status*)
		sStatTxt : STRING[200] := ''; (*User Folder's State in Text*)
		tyAlmData : tyAlmDat; (*Alarm Data*)
	END_STRUCT;
END_TYPE
```

### Program Logical/UsrFolder/UsrFolder (IEC, version 1.00.0) - 1.00.0 - NtFileIO v5.00.0 (2018-12-07)

#### Cyclic.st - Do Not Change!!!
```iecst
(** 2019-03-29 **)
PROGRAM _CYCLIC

	IF bInitialDone = FALSE THEN
		bInitialDone	:= TRUE;
		Act_Initial;
	ELSE
		Act_InputConfig;
		Act_Main;
		Act_OutputConfig;
		Act_Alarm;

	END_IF

END_PROGRAM
```

#### Act_Main.st - Do Not Change!!!
```iecst
(** 2019-05-09 **)
ACTION Act_Main:

	//Reset Done. Done Only Exist One Cycle.
	IF tylocalUsrFolder.Out.eStatus = Done AND tylocalUsrFolder.In.eAct = UsrFolderActIdle THEN
		tylocalUsrFolder.Out.eStat	:= UsrFolderActIdle;
	END_IF

	//Set tylocalUsrFolder.In.eAct
	IF tylocalUsrFolder.Out.eStatus = Idle THEN
		tylocalUsrFolder.Out.eStat	:= tylocalUsrFolder.In.eAct;
	END_IF
	//Main
	CASE tylocalUsrFolder.Out.eStat OF

		UsrFolderActIdle:
			IF tylocalUsrFolder.Out.eStatus <> Idle THEN	//Reset Data
				//Private
				fbDirCreate1(bEn := FALSE);
				fbDirCreate2(bEn := FALSE);
				fbDirCreate3(bEn := FALSE);
				fbDirCreate4(bEn := FALSE);

				tylocalUsrFolder.Out.sStatTxt	:= a_sStatText[tylocalUsrFolder.Out.eStat];

			END_IF

			tylocalUsrFolder.Out.eStatus	:= Idle;

		UsrFolderActCreateUsrDir:
			IF tylocalUsrFolder.Out.eStatus = Idle OR tylocalUsrFolder.Out.eStatus = Busy THEN

				tylocalUsrFolder.Out.eStatus	:= Busy;

				tylocalUsrFolder.Out.sStatTxt	:= a_sStatText[tylocalUsrFolder.Out.eStat];

				fbDirCreate1(bEn := TRUE);
				IF fbDirCreate1.udiStatus = 0 THEN
					tylocalUsrFolder.Out.eStatus		:= Done;
				ELSIF fbDirCreate1.udiStatus < 65534 THEN
					tylocalUsrFolder.Out.eStatus		:= Error;

					IF fbDirCreate1.udiStatus = 1908 THEN
						udiStatus	:= 10000;	//Creating User Directory Error
					ELSE
						udiStatus	:= fbDirCreate1.udiStatus;
					END_IF
				END_IF

			END_IF

		UsrFolderActCreatePrivateDir:
			IF tylocalUsrFolder.Out.eStatus = Idle OR tylocalUsrFolder.Out.eStatus = Busy THEN

				tylocalUsrFolder.Out.eStatus	:= Busy;

				tylocalUsrFolder.Out.sStatTxt	:= a_sStatText[tylocalUsrFolder.Out.eStat];

				fbDirCreate2(bEn := TRUE);
				IF fbDirCreate2.udiStatus = 0 THEN
					tylocalUsrFolder.Out.eStatus		:= Done;
				ELSIF fbDirCreate2.udiStatus < 65534 THEN
					tylocalUsrFolder.Out.eStatus		:= Error;

					IF fbDirCreate2.udiStatus = 1908 THEN
						udiStatus	:= 10001;	//Creating Private Directory Error
					ELSE
						udiStatus	:= fbDirCreate2.udiStatus;
					END_IF
				END_IF

			END_IF

		UsrFolderActCreateLogDir:
			IF tylocalUsrFolder.Out.eStatus = Idle OR tylocalUsrFolder.Out.eStatus = Busy THEN

				tylocalUsrFolder.Out.eStatus	:= Busy;

				tylocalUsrFolder.Out.sStatTxt	:= a_sStatText[tylocalUsrFolder.Out.eStat];

				fbDirCreate3(bEn := TRUE);
				IF fbDirCreate3.udiStatus = 0 THEN
					tylocalUsrFolder.Out.eStatus		:= Done;
				ELSIF fbDirCreate3.udiStatus < 65534 THEN
					tylocalUsrFolder.Out.eStatus		:= Error;

					IF fbDirCreate3.udiStatus = 1908 THEN
						udiStatus	:= 10002;	//Creating Log Directory Error
					ELSE
						udiStatus	:= fbDirCreate3.udiStatus;
					END_IF
				END_IF

			END_IF

		UsrFolderActCreateLCSDir:
			IF tylocalUsrFolder.Out.eStatus = Idle OR tylocalUsrFolder.Out.eStatus = Busy THEN

				tylocalUsrFolder.Out.eStatus	:= Busy;

				tylocalUsrFolder.Out.sStatTxt	:= a_sStatText[tylocalUsrFolder.Out.eStat];

				fbDirCreate4(bEn := TRUE);
				IF fbDirCreate4.udiStatus = 0 THEN
					tylocalUsrFolder.Out.eStatus		:= Done;
				ELSIF fbDirCreate4.udiStatus < 65534 THEN
					tylocalUsrFolder.Out.eStatus		:= Error;

					IF fbDirCreate4.udiStatus = 1908 THEN
						udiStatus	:= 10003;	//Creating LCS Directory Error
					ELSE
						udiStatus	:= fbDirCreate4.udiStatus;
					END_IF
				END_IF

			END_IF

	END_CASE

END_ACTION
```

#### Act_Alarm.st - Do Not Change!!!
```iecst
(** 2019-03-25 **)
ACTION Act_Alarm:

	IF tylocalUsrFolder.In.udiRstErr <> udiRstErrOld THEN
		bRstErr			:= TRUE;
		udiRstErrOld	:= tylocalUsrFolder.In.udiRstErr;
	ELSE
		bRstErr			:= FALSE;
	END_IF

	//Reset Error
	IF (tylocalUsrFolder.Out.eStatus = Error) AND bRstErr THEN
		tylocalUsrFolder.In.eAct	:= UsrFolderActIdle;
		tylocalUsrFolder.Out.eStat	:= UsrFolderActIdle;
	END_IF

	//Error
	IF EDGEPOS(tylocalUsrFolder.Out.eStatus = Error) THEN

		tyAlmData.sProgNm		:= p_sProgNm;
		tyAlmData.udiCode		:= udiStatus;
		tyAlmData.eSeverity		:= AlmSeverityError;
		tyAlmData.udiRunTime	:= tyAlmData.udiRunTime + 1;
		tyAlmData.bAlm			:= TRUE;
		tyAlmData.udiModuleNum  := udiModuleNum;
		g_sUsrFolderProgNm		:= p_sProgNm;

		//Get Error Message
		IF tyAlmData.udiCode < 10000 OR tyAlmData.udiCode > 10099 THEN
			tyAlmData.sAlmMsg	:= 'Unknown';
			tyAlmData.sRcyMsg	:= 'Unknown';
		ELSE
			tyAlmData.sAlmMsg	:= a_tyAlmText[tyAlmData.udiCode].sAlmText;
			tyAlmData.sRcyMsg	:= a_tyAlmText[tyAlmData.udiCode].sRcyText;
		END_IF

		tylocalUsrFolder.Out.sStatTxt	:= tyAlmData.sAlmMsg;

	ELSIF bRstErr AND (tyAlmData.udiCode <> 0) THEN

		tyAlmData.udiCode	:= 0;
		tyAlmData.eSeverity	:= AlmSeverityNA;
		tyAlmData.sAlmMsg	:= '';
		tyAlmData.sRcyMsg	:= '';
		tyAlmData.bAlm			:= FALSE;

		tylocalUsrFolder.Out.sStatTxt	:= a_sStatText[tylocalUsrFolder.Out.eStat];

	END_IF

END_ACTION
```

#### Local.var - Do Not Change!!!
```iecst
(*2019-05-09*)
(**)
(*Local Action, State & Status*)
VAR
	udiStatus : UDINT := 0;
	a_sStatText : ARRAY[0..50] OF STRING[200] := ['Idling','Creating User Directory','Creating Private Directory','Creating Log Directory','Creating LCS Directory',46('')];
END_VAR
(**)
(*Local Alarm*)
VAR
	tyAlmData : tyAlmDat;
	a_tyAlmText : ARRAY[10000..10099] OF tyAlmTxt := [(sAlmText:='Creating User Directory Error',sRcyText:='An Error Occured While Attempting To Create User Directory. Please Contact Nutek For A Possible Solution'),(sAlmText:='Creating Private Directory Error',sRcyText:='An Error Occured While Attempting To Create Private Directory. Please Contact Nutek For A Possible Solution'),(sAlmText:='Creating Log Directory Error',sRcyText:='An Error Occured While Attempting To Create Log Directory. Please Contact Nutek For A Possible Solution'),(sAlmText:='Creating LCS Directory Error',sRcyText:='An Error Occured While Attempting To Create LCS Directory. Please Contact Nutek For A Possible Solution'),96(0)];
END_VAR
(**)
(*Local Output*)
(**)
(*Local Input*)
VAR
	udiRstErr : UDINT := 0;
	sProgNm : STRING[15] := 'UsrFolder';
END_VAR
(**)
(*Local*)
VAR
	bRstErr : BOOL;
	udiRstErrOld : UDINT;
	bInitialDone : BOOL;
	fbDirCreate1 : fbDirCreate;
	fbDirCreate2 : fbDirCreate;
	fbDirCreate3 : fbDirCreate;
	fbDirCreate4 : fbDirCreate;
END_VAR
(**)
VAR
	udiModuleNum : UDINT := 5551;
END_VAR
```

#### Act_InputConfig.st - Change By Project
```iecst
ACTION Act_InputConfig:

	tylocalUsrFolder.In.udiRstErr := g_tyRstErrOut.udiRstErr;
	tylocalUsrFolder.In.eAct	  := g_tyStartUp.eUsrFolderAct;
	tylocalUsrFolder.In.sProgNm   := g_tyNtParamCurr.sUsrFolderProgNm;

END_ACTION
```

#### Act_OutputConfig.st - Change By Project
```iecst
ACTION Act_OutputConfig:

	g_tyUsrFolder := tylocalUsrFolder.Out;

END_ACTION
```

### Package Logical/LibVer - checked

### LibVer.typ - Do Not Change!!!
```iecst
(*2018-12-07*)
(**)
(*Action*)

TYPE
	eLibVerAction :
		(
		LibVerActIdle,
		LibVerActCreateDir,
		LibVerActWrite,
		LibVerActRead,
		LibVerActReadChk
		);
	tyLibVer : 	STRUCT
		In : tyLibVerIn1;
		Out : tyLibVerOut1;
	END_STRUCT;
	tyLibVerIn1 : 	STRUCT
		eAct : eLibVerAction; (*Library Version's Action*)
		udiRstErr : UDINT := 0; (*Reset Error*)
		a_tyInfoIn : ARRAY[0..c_diLibNum]OF tyLibrariesVer; (*Info Input*)
		sProgNm : STRING[15] := 'LibVer'; (*Program's Name*)
		bNtSettingsLoadDone : BOOL := TRUE; (*Nutek Parameters Settings Loading is Done*)
	END_STRUCT;
	tyLibVerOut1 : 	STRUCT
		eStat : eLibVerAction := LibVerActIdle; (*Library Version's State*)
		eStatus : eFBStatus := Idle; (*Library Versuib;s Status*)
		sStatTxt : STRING[200] := ''; (*Library Version's State in Text*)
		tyAlmData : tyAlmDat; (*Alarm Data*)
		a_tyInfoOut : ARRAY[0..c_diLibNum]OF tyLibrariesVer; (*Info Output [Array]*)
		a_bVerMismatch : ARRAY[0..c_diLibNum]OF BOOL; (*Version Mismatch [Array]*)
	END_STRUCT;
END_TYPE
```

### LibVer.var - Change By Project
```iecst
(*2019-03-25*)
VAR
	g_tyLibVer : tyLibVerOut1;
END_VAR
(**)
(**)
(*Alarm*)
VAR
	p_LibVerAlmData : UDINT;
END_VAR
(**)
(*Output*)
VAR
	p_LibVerInfoOut : UDINT;
	p_VerMismatch : UDINT;
END_VAR
```

### Program Logical/LibVer/LibVer (IEC, version 1.00.0) - 1.00.0 - NtVersion v5.00.0 , NtFileIO v5.00.0 (2018-12-07)

#### Cyclic.st - Do Not Change!!!
```iecst
(** 2019-03-29 **)
PROGRAM _CYCLIC

	IF bInitialDone = FALSE THEN
		IF g_tyStartUp.bNtSettingsLoadDone = TRUE THEN
			bInitialDone	:= TRUE;

			Act_Initial;
		END_IF

	ELSE
		Act_InputConfig;
		Act_Main;
		Act_OutputConfig;
		Act_Alarm;

	END_IF

END_PROGRAM
```

#### Act_Initial.st - Do Not Change!!!
```iecst
ACTION Act_Initial:

	//Initial
	tylocalLibVer.Out.sStatTxt	:= a_sStatText[tylocalLibVer.Out.eStat];

	fbDirCreate1.sDevice	:= 'C';
	fbDirCreate1.sDirName	:= 'User';
	fbDirCreate1(bEn := FALSE);

	fbDirCreate2.sDevice	:= 'User';
	fbDirCreate2.sDirName	:= 'LibrariesVersion';
	fbDirCreate2(bEn := FALSE);

	fbFileRead1.sDevice		:= 'LibVer';
	fbFileRead1.sFile		:= 'LibrariesVersion.dat';
	fbFileRead1.udiOffset	:= 0;
	fbFileRead1.p_Dest		:= ADR(tylocalLibVer.Out.a_tyInfoOut);
	fbFileRead1.udiLen		:= SIZEOF(tylocalLibVer.Out.a_tyInfoOut);
	fbFileRead1(bEn := FALSE);

	fbFileWrite1.sDevice	:= 'LibVer';
	fbFileWrite1.sFile		:= 'LibrariesVersion.dat';
	fbFileWrite1.udiOffset	:= 0;
	fbFileWrite1.p_Src		:= ADR(tylocalLibVer.In.a_tyInfoIn);
	fbFileWrite1.udiLen		:= SIZEOF(tylocalLibVer.In.a_tyInfoIn);
	fbFileWrite1.udiOption	:= 0;
	fbFileWrite1(bEn := FALSE);

	fbChkLibVerFile(bEn := FALSE);

	fbChkLibVer.pa_bVerMismatch := ADR(tylocalLibVer.Out.a_bVerMismatch);
	fbChkLibVer(bEn := FALSE);

END_ACTION
```

#### Act_Main.st - Do Not Change!!!
```iecst
(** 2020-08-17 **)
ACTION Act_Main:

	//Reset Done
	IF tylocalLibVer.Out.eStatus = Done AND tylocalLibVer.In.eAct = LibVerActIdle THEN
		tylocalLibVer.Out.eStat	:= LibVerActIdle;
	END_IF

	//Set p_eAct
	IF tylocalLibVer.Out.eStatus = Idle THEN
		tylocalLibVer.Out.eStat	:= p_eAct;
	END_IF
	//Main
	CASE tylocalLibVer.Out.eStat OF

		LibVerActIdle:
			IF tylocalLibVer.Out.eStatus <> Idle THEN	//Reset Data
				//Private
				fbDirCreate1(bEn := FALSE);
				fbDirCreate2(bEn := FALSE);
				fbFileRead1(bEn := FALSE);
				fbFileWrite1(bEn := FALSE);
				fbChkLibVerFile(bEn := FALSE);
				fbChkLibVer(bEn := FALSE);
				usiStep	:= 0;
				memset(ADR(a_bVerMismatch), 0, SIZEOF(a_bVerMismatch));

				tylocalLibVer.Out.sStatTxt	:= a_sStatText[tylocalLibVer.Out.eStat];

			END_IF

			tylocalLibVer.Out.eStatus	:= Idle;

		LibVerActCreateDir:
			IF tylocalLibVer.Out.eStatus = Idle OR tylocalLibVer.Out.eStatus = Busy THEN

				tylocalLibVer.Out.eStatus	:= Busy;

				tylocalLibVer.Out.sStatTxt	:= a_sStatText[tylocalLibVer.Out.eStat];

				CASE usiStep OF
					0:
						fbDirCreate1(bEn := TRUE);
						IF fbDirCreate1.udiStatus = 0 THEN
							usiStep	:= 1;
						ELSIF fbDirCreate1.udiStatus < 65534 THEN
							tylocalLibVer.Out.eStatus		:= Error;

							IF fbDirCreate1.udiStatus = 1908 THEN
								udiStatus	:= 10000;	//Creating Private Directory Error
							ELSE
								udiStatus	:= fbDirCreate1.udiStatus;
							END_IF
						END_IF

					1:
						fbDirCreate2(bEn := TRUE);
						IF fbDirCreate2.udiStatus = 0 THEN
							tylocalLibVer.Out.eStatus	:= Done;
						ELSIF fbDirCreate2.udiStatus < 65534 THEN
							tylocalLibVer.Out.eStatus		:= Error;

							IF fbDirCreate2.udiStatus = 1908 THEN
								udiStatus	:= 10001;	//Creating User Management Directory Error
							ELSE
								udiStatus	:= fbDirCreate2.udiStatus;
							END_IF
						END_IF

				END_CASE

			END_IF

		LibVerActWrite:
			IF tylocalLibVer.Out.eStatus = Idle OR tylocalLibVer.Out.eStatus = Busy THEN

				tylocalLibVer.Out.eStatus	:= Busy;

				tylocalLibVer.Out.sStatTxt	:= a_sStatText[tylocalLibVer.Out.eStat];

				fbFileWrite1(bEn := TRUE);

				IF fbFileWrite1.udiStatus = 0 THEN
					tylocalLibVer.Out.eStatus	:= Done;
				ELSIF fbFileWrite1.udiStatus < 65534 THEN
					tylocalLibVer.Out.eStatus			:= Error;

					IF fbFileWrite1.udiStatus = 1900 THEN
						udiStatus	:= 10002;	//File Open Error While Writing
					ELSIF fbFileWrite1.udiStatus = 1901 THEN
						udiStatus	:= 10003;	//File Create Error While Writing
					ELSIF fbFileWrite1.udiStatus = 1903 THEN
						udiStatus	:= 10004;	//File Write Error
					ELSIF fbFileWrite1.udiStatus = 1904 THEN
						udiStatus	:= 10005;	//File Close Error While Writing
					ELSIF fbFileWrite1.udiStatus = 1914 THEN
						udiStatus	:= 10013;	//Directory Does Not Exist While Writing
					ELSE
						udiStatus	:= fbFileWrite1.udiStatus;
					END_IF
				END_IF

			END_IF

		LibVerActRead:
			IF tylocalLibVer.Out.eStatus = Idle OR tylocalLibVer.Out.eStatus = Busy THEN

				tylocalLibVer.Out.eStatus	:= Busy;

				tylocalLibVer.Out.sStatTxt	:= a_sStatText[tylocalLibVer.Out.eStat];

				fbFileRead1(bEn := TRUE);
				IF fbFileRead1.udiStatus = 0 THEN
					tylocalLibVer.Out.eStatus	:= Done;
				ELSIF fbFileRead1.udiStatus < 65534 THEN
					tylocalLibVer.Out.eStatus		:= Error;

					IF fbFileRead1.udiStatus = 1900 THEN
						udiStatus	:= 10006;	//File Open Error While Reading
					ELSIF fbFileRead1.udiStatus = 1902 THEN
						udiStatus	:= 10007;	//File Read Error
					ELSIF fbFileRead1.udiStatus = 1904 THEN
						udiStatus	:= 10008;	//File Close Error While Reading
					ELSIF fbFileRead1.udiStatus = 1915 THEN
						udiStatus	:= 10014;	//File Not Found While Reading
					ELSE
						udiStatus	:= fbFileRead1.udiStatus;
					END_IF
				END_IF

			END_IF

		LibVerActReadChk:
			IF tylocalLibVer.Out.eStatus = Idle OR tylocalLibVer.Out.eStatus = Busy THEN

				tylocalLibVer.Out.eStatus	:= Busy;

				tylocalLibVer.Out.sStatTxt	:= a_sStatText[tylocalLibVer.Out.eStat];

				CASE usiStep OF
					0:
						fbFileRead1(bEn := TRUE);
						IF fbFileRead1.udiStatus = 0 THEN
							usiStep	:= 1;
						ELSIF fbFileRead1.udiStatus < 65534 THEN
							tylocalLibVer.Out.eStatus		:= Error;

							IF fbFileRead1.udiStatus = 1900 THEN
								udiStatus	:= 10009;	//File Open Error While Checking
							ELSIF fbFileRead1.udiStatus = 1902 THEN
								udiStatus	:= 10010;	//File Read Error While Checking
							ELSIF fbFileRead1.udiStatus = 1904 THEN
								udiStatus	:= 10011;	//File Close Error While Checking
							ELSIF fbFileRead1.udiStatus = 1915 THEN
								udiStatus	:= 10015;	//File Not Found While Checking
							ELSE
								udiStatus	:= fbFileRead1.udiStatus;
							END_IF
						END_IF

					1:
						fbChkLibVerFile.a_tyLibraryVer := a_tyInfoOut;

						fbChkLibVerFile(bEn := TRUE);
						IF fbChkLibVerFile.udiStatus = 0 THEN
							usiStep	:= 2;
						ELSIF fbChkLibVerFile.udiStatus < 65534 THEN
							tylocalLibVer.Out.eStatus		:= Error;

							IF fbChkLibVerFile.udiStatus = 1001 THEN
								udiStatus	:= 10016;	//Libraries Version File Corrupted
							END_IF
						END_IF

					2:

						fbChkLibVer.a_tyLibraryVer := a_tyInfoOut;

						fbChkLibVer(bEn := TRUE);
						IF fbChkLibVer.udiStatus = 0 THEN
							tylocalLibVer.Out.eStatus	:= Done;
						ELSIF fbChkLibVer.udiStatus < 65534 THEN
							tylocalLibVer.Out.eStatus		:= Error;

							IF fbChkLibVer.udiStatus = 1002 THEN
								udiStatus	:= 10012;	//Libraries Version Mismatch
							END_IF
						END_IF

				END_CASE

			END_IF

	END_CASE

END_ACTION
```

#### Act_Alarm.st - Do Not Change!!!
```iecst
(** 2019-03-25 **)
ACTION Act_Alarm:
	IF tylocalLibVer.In.udiRstErr <> udiRstErrOld THEN
		bRstErr			:= TRUE;
		udiRstErrOld	:= tylocalLibVer.In.udiRstErr;
	ELSE
		bRstErr			:= FALSE;
	END_IF

	//Reset Error
	IF (tylocalLibVer.Out.eStatus = Error) AND bRstErr THEN
		tylocalLibVer.In.eAct	:= LibVerActIdle;
		tylocalLibVer.Out.eStat	:= LibVerActIdle;

	END_IF

	//Error
	IF EDGEPOS(tylocalLibVer.Out.eStatus = Error) THEN

		tylocalLibVer.Out.tyAlmData.udiCode		:= udiStatus;
		tylocalLibVer.Out.tyAlmData.udiRunTime	:= tylocalLibVer.Out.tyAlmData.udiRunTime + 1;
		g_tyAlmProgNm.sLibVerProgNm				:= tylocalLibVer.In.sProgNm;

		IF tylocalLibVer.Out.tyAlmData.udiCode = 10012 THEN
			tylocalLibVer.Out.tyAlmData.eSeverity	:= AlmSeverityWarning;
			tylocalLibVer.Out.tyAlmData.bWarning		:= TRUE;

			FOR di := 0 TO c_diLibNum DO
				IF a_bVerMismatch[di] = TRUE THEN
					g_tyAlmProgNm.sLiberWarnName    := a_tyInfoOut[di].sName;
					EXIT;
				END_IF
			END_FOR

		ELSE
			tylocalLibVer.Out.tyAlmData.eSeverity	:= AlmSeverityError;
			tylocalLibVer.Out.tyAlmData.bAlm		:= TRUE;

		END_IF

	ELSIF bRstErr AND (tylocalLibVer.Out.tyAlmData.udiCode <> 0) THEN

		tylocalLibVer.Out.tyAlmData.udiCode	:= 0;
		tylocalLibVer.Out.tyAlmData.eSeverity	:= AlmSeverityNA;
		tylocalLibVer.Out.tyAlmData.bAlm		:= FALSE;
		tylocalLibVer.Out.tyAlmData.bWarning	:= FALSE;

		tylocalLibVer.Out.sStatTxt	:= a_sStatText[tylocalLibVer.Out.eStat];

	END_IF

END_ACTION
```

#### Act_InputConfig.st - not listed in the package file held
```iecst
ACTION Act_InputConfig:

	tylocalLibVer.In.udiRstErr := g_tyRstErrOut.udiRstErr;
	tylocalLibVer.In.eAct	   := g_tyStartUp.eLibVerAct;
	tylocalLibVer.In.sProgNm   := g_tyNtParamCurr.sLibVersionProgNm;

END_ACTION
```

#### Act_OutputConfig.st - not listed in the package file held
```iecst
ACTION Act_OutputConfig:

	g_tyLibVer := tylocalLibVer.Out;

END_ACTION
```

### Time.typ - Do Not Change!!!
```iecst
TYPE
	eTimeAction :
		(
		TimeActIdle,
		TimeActGetTime,
		TimeActGetTimeZone,
		TimeActSetTime,
		TimeActSetTimeZone
		);
	tyTime : 	STRUCT
		In : tyTimeIn1;
		Out : tyTimeOut1;
	END_STRUCT;
	tyTimeIn1 : 	STRUCT
		eAct : eTimeAction; (*Time's Action*)
		udiRstErr : UDINT := 0; (*Reset Error*)
		dtSetDT : DATE_AND_TIME; (*Set Date Time*)
		uiSetTimeZone : UINT; (*Set Time Zone*)
		sProgNm : STRING[15] := 'Time'; (*Program's Name*)
		bNtSettingsLoadDone : BOOL := TRUE; (*Nutek Parameter Setting Loading is Done*)
	END_STRUCT;
	tyTimeOut1 : 	STRUCT
		eStat : eTimeAction := TimeActIdle; (*Time's State*)
		eMainStatus : eFBStatus := Idle; (*Time's Status*)
		sStatTxt : STRING[200] := ''; (*Time's State in Text*)
		tyAlmData : tyAlmDat; (*Alarm Data*)
		tyAlmData1 : tyAlmDat; (*Alarm Data 1*)
		dtCurrDT : DATE_AND_TIME; (*Current Date Time*)
		uiCurrTimeZone : UINT; (*Current Time Zone*)
		tyCurrDTStruct : DTStructure; (*Current Date Time Structure*)
	END_STRUCT;
END_TYPE
```

### Time.var - Change By Project
```iecst
VAR
	g_tyTime : tyTimeOut1;
END_VAR
```

### Program Logical/Time/Time (IEC, version 1.00.0) - 1.00.0 - 

#### Init.st - Change By Project
```iecst
(** 2019-03-25 **)
PROGRAM _INIT

	(* Always Change If Project Change *)

	//Pass Address To Global Address For External Use
	//Action, State & Status
	p_TimeStat		:= ADR(eStat);
	p_TimeStatus	:= ADR(eMainStatus);
	p_TimeStatTxt	:= ADR(sStatTxt);

	//Alarm
	p_TimeAlmData	:= ADR(tyAlmData);
	p_TimeAlmData1	:= ADR(tyAlmData1);

	//Output
	p_TimeCurrDT		:= ADR(dtCurrDT);
	p_TimeCurrTimeZone	:= ADR(uiCurrTimeZone);
	p_TimeCurrDTStruct	:= ADR(tyCurrDTStruct);
	p_TimeCurrDTStructMS := ADR(tyCurrDTStruct.millisec);
	(* Always Change If Project Change *)

END_PROGRAM
```

#### Cyclic.st - Do Not Change!!!
```iecst
PROGRAM _CYCLIC

	IF bInitialDone = FALSE THEN
		IF g_tyStartUp.bNtSettingsLoadDone = TRUE THEN
			bInitialDone	:= TRUE;
			Act_Initial;
		END_IF

	ELSE

		Act_InputConfig;
		Act_Main;
		Act_OutputConfig;
		Act_Alarm;

	END_IF

END_PROGRAM
```

#### Act_Initial.st - Do Not Change!!!
```iecst
ACTION Act_Initial:

	//Initial
	tylocalTime.Out.sStatTxt	:= a_sStatText[tylocalTime.Out.eStat];

	fbSetTime(enable := FALSE);

	fbSetTimeZone.option	:= cfgOPTION_NON_VOLATILE;
	fbSetTimeZone(enable := FALSE);

	fbGetTime(enable := FALSE);

	fbGetTime1(enable := FALSE);

	fbGetTimeDT.pDTStructure	:= ADR(tylocalTime.Out.tyCurrDTStruct);
	fbGetTimeDT(enable := FALSE);

	fbGetTimeDT1.pDTStructure	:= ADR(tylocalTime.Out.tyCurrDTStruct);
	fbGetTimeDT1(enable := FALSE);

	fbGetTimeZone(enable := FALSE);

	fbDlyTm(IN := FALSE);

END_ACTION
```

#### Act_Main.st - Do Not Change!!!
```iecst
ACTION Act_Main:

	IF (eStatus1 = Error) AND bRstErr THEN
		eStatus1	:= Idle;
		udiStatus1	:= 0;
		fbDlyTm(IN := FALSE);
		fbGetTime1(enable := FALSE);
		fbGetTimeDT1(enable := FALSE);
	END_IF

	IF eStatus1 <> Error THEN

		fbDlyTm(IN := TRUE);

		IF fbDlyTm.Q = TRUE THEN

			fbGetTime1(enable := TRUE);
			fbGetTimeDT1(enable := TRUE);

			IF fbGetTime1.status = 0 AND fbGetTimeDT1.status = 0 THEN
				tylocalTime.Out.dtCurrDT	:= fbGetTime1.DT1;
				fbGetTime1(enable := FALSE);
				fbGetTimeDT1(enable := FALSE);
				fbDlyTm(IN := FALSE);
			ELSIF fbGetTime1.status > 0 AND fbGetTime1.status < 65534 THEN
				udiStatus1	:= 5856;	//Get Time Error In Background
				eStatus1	:= Error;
			ELSIF fbGetTimeDT1.status > 0 AND fbGetTimeDT1.status < 65534 THEN
				udiStatus1	:= 5857;	//Get Time Structure Error In Background
				eStatus1	:= Error;
			END_IF

		END_IF

	END_IF

	//Reset Done
	IF eStatus = Done AND tylocalTime.In.eAct = TimeActIdle THEN
		tylocalTime.Out.eStat	:= TimeActIdle;
	END_IF
	//Set tylocalTime.In.eAct
	IF eStatus = Idle THEN
		tylocalTime.Out.eStat	:= tylocalTime.In.eAct;
	END_IF

	//Main
	CASE tylocalTime.Out.eStat OF

		TimeActIdle:
			IF eStatus <> Idle THEN	//Reset Data
				//Private
				fbSetTime(enable := FALSE);
				fbSetTimeZone(enable := FALSE);
				fbGetTime(enable := FALSE);
				fbGetTimeDT(enable := FALSE);
				fbGetTimeZone(enable := FALSE);

				tylocalTime.Out.sStatTxt	:= a_sStatText[tylocalTime.Out.eStat];

			END_IF

			eStatus	:= Idle;

		TimeActSetTime:
			IF eStatus = Idle OR eStatus = Busy THEN

				eStatus	:= Busy;

				tylocalTime.Out.sStatTxt	:= a_sStatText[tylocalTime.Out.eStat];

				fbSetTime.DT1	:= tylocalTime.In.dtSetDT;
				fbSetTime(enable := TRUE);

				IF fbSetTime.status = 0 THEN
					eStatus	:= Done;
				ELSIF fbSetTime.status < 65534 THEN
					udiStatus	:= 5851;	//Set Time Error
					eStatus		:= Error;
				END_IF

			END_IF

		TimeActSetTimeZone:
			IF eStatus = Idle OR eStatus = Busy THEN

				eStatus	:= Busy;

				tylocalTime.Out.sStatTxt	:= a_sStatText[tylocalTime.Out.eStat];

				fbSetTimeZone.timezoneID	:= tylocalTime.In.uiSetTimeZone;
				fbSetTimeZone(enable := TRUE);

				IF fbSetTimeZone.status = 0 THEN
					eStatus	:= Done;
				ELSIF fbSetTimeZone.status < 65534 THEN
					udiStatus	:= 5852;	//Set Time Zone Error
					eStatus		:= Error;
				END_IF

			END_IF

		TimeActGetTime:
			IF eStatus = Idle OR eStatus = Busy THEN

				eStatus	:= Busy;

				tylocalTime.Out.sStatTxt	:= a_sStatText[tylocalTime.Out.eStat];

				fbGetTime(enable := TRUE);
				fbGetTimeDT(enable := TRUE);

				IF fbGetTime.status = 0 AND fbGetTimeDT.status = 0 THEN
					tylocalTime.Out.dtCurrDT	:= fbGetTime.DT1;
					eStatus		:= Done;
				ELSIF fbGetTime.status > 0 AND fbGetTime.status < 65534 THEN
					udiStatus	:= 5853;	//Get Time Error
					eStatus		:= Error;
				ELSIF fbGetTimeDT.status > 0 AND fbGetTimeDT.status < 65534 THEN
					udiStatus	:= 5854;	//Get Time Structure Error
					eStatus		:= Error;
				END_IF

			END_IF

		TimeActGetTimeZone:
			IF eStatus = Idle OR eStatus = Busy THEN

				eStatus	:= Busy;

				tylocalTime.Out.sStatTxt	:= a_sStatText[tylocalTime.Out.eStat];

				fbGetTimeZone(enable := TRUE);

				IF fbGetTimeZone.status = 0 THEN
					tylocalTime.Out.uiCurrTimeZone	:= fbGetTimeZone.timezoneID;
					eStatus			:= Done;
				ELSIF fbGetTimeZone.status < 65534 THEN
					udiStatus	:= 5855;	//Get Time Zone Error
					eStatus		:= Error;
				END_IF

			END_IF

	END_CASE

	IF eStatus = Error OR eStatus1 = Error THEN
		tylocalTime.Out.eMainStatus	:= Error;
	ELSE
		tylocalTime.Out.eMainStatus	:= eStatus;
	END_IF

END_ACTION
```

#### Act_Alarm.st - Do Not Change!!!
```iecst
ACTION Act_Alarm:

	IF tylocalTime.In.udiRstErr <> udiRstErrOld THEN
		bRstErr			:= TRUE;
		udiRstErrOld	:= tylocalTime.In.udiRstErr;
	ELSE
		bRstErr			:= FALSE;
	END_IF

	IF (eStatus = Error) AND bRstErr THEN
		tylocalTime.In.eAct	:= TimeActIdle;
		tylocalTime.Out.eStat	:= TimeActIdle;
	END_IF

	//Error
	IF EDGEPOS(eStatus = Error) THEN

		tylocalTime.Out.tyAlmData.udiCode		:= udiStatus;
		tylocalTime.Out.tyAlmData.eSeverity		:= AlmSeverityError;
		tylocalTime.Out.tyAlmData.udiRunTime	:= tylocalTime.Out.tyAlmData.udiRunTime + 1;
		tylocalTime.Out.tyAlmData.bAlm			:= TRUE;
		tylocalTime.Out.tyAlmData.udiModuleNum  := udiModuleNum;
		g_tyAlmProgNm.sTimeProgNm				:= tylocalTime.In.sProgNm;

	ELSIF bRstErr AND (tylocalTime.Out.tyAlmData.udiCode <> 0) THEN

		tylocalTime.Out.tyAlmData.udiCode	:= 0;
		tylocalTime.Out.tyAlmData.eSeverity	:= AlmSeverityNA;
		tylocalTime.Out.tyAlmData.bAlm		:= FALSE;

		tylocalTime.Out.sStatTxt	:= a_sStatText[tylocalTime.Out.eStat];

	END_IF

	//Error
	IF EDGEPOS(eStatus1 = Error) THEN

		tylocalTime.Out.tyAlmData1.udiCode		:= udiStatus1;
		tylocalTime.Out.tyAlmData1.eSeverity	:= AlmSeverityError;
		tylocalTime.Out.tyAlmData1.udiRunTime	:= tylocalTime.Out.tyAlmData1.udiRunTime + 1;

		tylocalTime.Out.tyAlmData1.bAlm			:= TRUE;
		tylocalTime.Out.tyAlmData1.udiModuleNum := udiModuleNum;
		g_tyAlmProgNm.sTimeProgNm				:= tylocalTime.In.sProgNm;

	ELSIF bRstErr AND (tylocalTime.Out.tyAlmData1.udiCode <> 0) THEN

		tylocalTime.Out.tyAlmData1.udiCode		:= 0;
		tylocalTime.Out.tyAlmData1.eSeverity	:= AlmSeverityNA;
		tylocalTime.Out.tyAlmData1.bAlm			:= FALSE;

		tylocalTime.Out.sStatTxt	:= a_sStatText[tylocalTime.Out.eStat];

	END_IF

END_ACTION
```

#### Act_Alarm1.st - Do Not Change!!!
```iecst
(** 2019-03-25 **)
ACTION Act_Alarm1:

	//Error
	IF EDGEPOS(eStatus1 = Error) THEN

		tyAlmData1.sProgNm		:= p_sProgNm;
		tyAlmData1.udiCode		:= udiStatus1;
		tyAlmData1.eSeverity	:= AlmSeverityError;
		tyAlmData1.udiRunTime	:= tyAlmData1.udiRunTime + 1;
		tyAlmData1.bAlm			:= TRUE;
		tyAlmData1.udiModuleNum  := udiModuleNum;
		g_sTimeProgNm			:= p_sProgNm;

		//Get Error Message
		IF tyAlmData1.udiCode < 10000 OR tyAlmData1.udiCode > 10099 THEN
			tyAlmData1.sAlmMsg	:= 'Unknown';
			tyAlmData1.sRcyMsg	:= 'Unknown';
		ELSE
			tyAlmData1.sAlmMsg	:= a_tyAlmText[tyAlmData1.udiCode].sAlmText;
			tyAlmData1.sRcyMsg	:= a_tyAlmText[tyAlmData1.udiCode].sRcyText;
		END_IF

		sStatTxt	:= tyAlmData1.sAlmMsg;

	ELSIF bRstErr AND (tyAlmData1.udiCode <> 0) THEN

		tyAlmData1.udiCode		:= 0;
		tyAlmData1.eSeverity	:= AlmSeverityNA;
		tyAlmData1.sAlmMsg		:= '';
		tyAlmData1.sRcyMsg		:= '';
		tyAlmData1.bAlm			:= FALSE;
		sStatTxt	:= a_sStatText[eStat];

	END_IF

END_ACTION
```

#### Local.var - Do Not Change!!!
```iecst
VAR
	tylocalTime : tyTime;
	eStatus : eFBStatus := Idle;
	eStatus1 : eFBStatus := Idle;
	udiStatus : UDINT := 0;
	udiStatus1 : UDINT := 0;
	sStatTxt : STRING[200] := '';
	a_sStatText : ARRAY[0..50] OF STRING[200] := ['Idling','Get Time','Get Time Zone','Setting Time','Setting Time Zone',46('')];
	tyAlmData : tyAlmDat;
	tyAlmData1 : tyAlmDat;
END_VAR
(**)
(**)
VAR
	dtCurrDT : DATE_AND_TIME;
	uiCurrTimeZone : UINT;
	tyCurrDTStruct : DTStructure;
END_VAR
(**)
(**)
VAR
	udiRstErr : UDINT := 0;
	dtSetDT : DATE_AND_TIME;
	uiSetTimeZone : UINT;
	udiModuleNum : UDINT := 5851;
END_VAR
(*Local*)
VAR
	bRstErr : BOOL;
	udiRstErrOld : UDINT;
	bInitDone : BOOL;
	bInitialDone : BOOL;
	fbDlyTm : TON := (PT:=T#500ms);
	fbGetTime : DTGetTime;
	fbGetTime1 : DTGetTime;
	fbSetTime : DTSetTime;
	fbGetTimeDT : DTStructureGetTime;
	fbGetTimeDT1 : DTStructureGetTime;
	fbGetTimeZone : CfgGetTimeZone;
	fbSetTimeZone : CfgSetTimeZone;
	p_tyLFFollower : REFERENCE TO tyLFFollowerOut1;
END_VAR
```

#### Act_InputConfig.st - not listed in the package file held
```iecst
ACTION Act_InputConfig:

	p_tyLFFollower ACCESS p_LFFollower;

	tylocalTime.In.eAct 		:= p_tyLFFollower.eTimeAct;
	tylocalTime.In.dtSetDT		:= p_tyLFFollower.dtTm;
	tylocalTime.In.udiRstErr	:= g_tyRstErrOut.bSafetyRlyRst;
	tylocalTime.In.sProgNm		:= g_tyNtParamCurr.sTimeProgNm;

END_ACTION
```

#### Act_OutputConfig.st - not listed in the package file held
```iecst
ACTION Act_OutputConfig:

	g_tyTime := tylocalTime.Out;

END_ACTION
```

### HWInfo.typ - Do Not Change!!!
```iecst
(*2020-09-22*)
(**)
(*Action*)

TYPE
	eHWInfoAction :
		(
		HWInfoActIdle,
		HWInfoActGetIPAddr,
		HWInfoActGetSubnetMask,
		HWInfoActGetMacAddr,
		HWInfoActSetIPAddr,
		HWInfoActSetSubnetMask,
		HWInfoActGetEthConfigMode,
		HWInfoActSetEthConfigMode,
		HWInfoActSetDefaultGateway
		);
	eNetworkConfigMod :
		(
		SetIPManually := 0,
		IPFromDHCPServer := 1
		);
	tysMacAddress : 	STRUCT
		s_PLCMacAddr0 : STRING[2];
		s_PLCMacAddr1 : STRING[2];
		s_PLCMacAddr2 : STRING[2];
		s_PLCMacAddr3 : STRING[2];
		s_PLCMacAddr4 : STRING[2];
		s_PLCMacAddr5 : STRING[2];
	END_STRUCT;
END_TYPE

(*Action*)

TYPE
	tyHWInfo : 	STRUCT
		In : tyHWInfoIn1;
		Out : tyHWInfoOut1;
	END_STRUCT;
	tyHWInfoIn1 : 	STRUCT
		eAct : eHWInfoAction; (*Hardware Info's Action*)
		udiRstErr : UDINT := 0; (*Reset Error*)
		sSetIPAddr : STRING[15]; (*Set IP Address*)
		sSetSubnetMask : STRING[15]; (*Set Subnet Mask*)
		sDevice : STRING[3] := 'IF2'; (*Device's Name*)
		sProgNm : STRING[15] := 'HWInfo'; (*Program's Name*)
		bNtSettingsLoadDone : BOOL := TRUE; (*Nutek Parameter Settings Loading is Done*)
		usiNetworkMode : USINT; (*Network Mode*)
		sHMIMacAdd : STRING[27];
		sSetDefaultGW : STRING[15];
	END_STRUCT;
	tyHWInfoOut1 : 	STRUCT
		eStat : eHWInfoAction := HWInfoActIdle; (*Hardware Info's State*)
		eStatus : eFBStatus := Idle; (*Hardware Info's Status*)
		sStatTxt : STRING[200] := ''; (*Hardware Info's State in Text*)
		tyAlmData : tyAlmDat; (*Alarm Data*)
		sIPAddr : STRING[15]; (*IP Address*)
		sSubnetMask : STRING[15]; (*Subnet Mask*)
		a_usiMacAddr : ARRAY[0..5]OF USINT; (*Mac Address*)
		udiConfigMode : UDINT; (*Configuration Mode*)
	END_STRUCT;
END_TYPE
```

### HWInfo.var - Change By Project
```iecst
(*2020-09-22*)
VAR
	g_tyHWInfo : tyHWInfoOut1;
END_VAR
(**)
(*Action & State & Status*)
VAR
	p_HWInfoStat : UDINT;
	p_HWInfoStatus : UDINT;
	p_HWInfoStatTxt : UDINT;
END_VAR
(**)
(*Alarm*)
VAR
	p_HWInfoAlmData : UDINT;
END_VAR
(**)
(*Output*)
VAR
	p_HWInfoIPAddr : UDINT;
	p_HWInfoMacAddr : UDINT;
	p_HWInfoSubnetMask : UDINT;
	p_HWInfoEthMode : UDINT;
END_VAR
```

### Program Logical/HWInfo/HWInfo (IEC, version 1.00.0) - 1.00.0 - 

#### Act_InputConfig.st - Change By Project
```iecst
ACTION Act_InputConfig:

	tylocalHWInfo.In.udiRstErr 		:= g_tyRstErrOut.udiRstErr;
	tylocalHWInfo.In.sSetIPAddr		:= g_tyUIOut.sSetIPAddr;
	tylocalHWInfo.In.sSetSubnetMask	:= g_tyUIOut.sSetSubnetMask;
	tylocalHWInfo.In.sDevice		:= g_tyNtParamCurr.sHWInfoDevice;
	tylocalHWInfo.In.sProgNm		:= g_tyNtParamCurr.sHWInfoProgNm;
	tylocalHWInfo.In.usiNetworkMode	:= g_tyUIOut.usiNetworkModeSelected;
	tylocalHWInfo.In.sHMIMacAdd		:= g_tyNtParamCurr.sHWInfoHMIMacAddress;
	tylocalHWInfo.In.sSetDefaultGW	:= g_tyMcParamCurr.sDefaultGateWay;

	IF g_tyStartUp.bRun THEN
		tylocalHWInfo.In.eAct := g_tyStartUp.eHWInfoAct;
	ELSE
		tylocalHWInfo.In.eAct := g_tyUIOut.eMnlAct.eHWInfoAct;
	END_IF

END_ACTION
```

#### Act_OutputConfig.st - Change By Project
```iecst
ACTION Act_OutputConfig:

	g_tyHWInfo := tylocalHWInfo.Out;

END_ACTION
```

#### Act_Link.st - Change By Project
```iecst
(** 2019-03-29 **)
ACTION Act_Link:

	// PLC MAC Address
	fConvertUSINTToHex (ADR(sMacAddress.s_PLCMacAddr0),(a_usiMacAddr[0]));
	fConvertUSINTToHex (ADR(sMacAddress.s_PLCMacAddr1),(a_usiMacAddr[1]));
	fConvertUSINTToHex (ADR(sMacAddress.s_PLCMacAddr2),(a_usiMacAddr[2]));
	fConvertUSINTToHex (ADR(sMacAddress.s_PLCMacAddr3),(a_usiMacAddr[3]));
	fConvertUSINTToHex (ADR(sMacAddress.s_PLCMacAddr4),(a_usiMacAddr[4]));
	fConvertUSINTToHex (ADR(sMacAddress.s_PLCMacAddr5),(a_usiMacAddr[5]));

	//Combine PLC MAC Address
	sPLCMacAddress	:= CONCAT(CONCAT(CONCAT(CONCAT(CONCAT(CONCAT(sMacAddress.s_PLCMacAddr0,' - '),CONCAT(sMacAddress.s_PLCMacAddr1,' - ')),CONCAT(sMacAddress.s_PLCMacAddr2,' - ')),CONCAT(sMacAddress.s_PLCMacAddr3,' - ')),CONCAT(sMacAddress.s_PLCMacAddr4,' - ')),sMacAddress.s_PLCMacAddr5);

	//HMI Mac Address
	sHMIMacAddress	:= p_sHMIMacAdd;
END_ACTION
```

#### Cyclic.st - Do Not Change!!!
```iecst
(** 2019-03-29 **)
PROGRAM _CYCLIC

	IF bInitialDone = FALSE THEN
		IF p_bNtSettingsLoadDone = TRUE THEN
			bInitialDone	:= TRUE;
			Act_Initial;
		END_IF

	ELSE
		Act_InputConfig;
		Act_Link;
		Act_Main;
		Act_OutputConfig;
		Act_Alarm;

	END_IF

END_PROGRAM
```

#### Act_Initial.st - Do Not Change!!!
```iecst
(** 2020-09-22 **)
ACTION Act_Initial:

	//Initial
	sStatTxt	:= a_sStatText[eStat];

	fbGetIPAddr.pDevice	:= ADR(p_sDevice);
	fbGetIPAddr.pIPAddr	:= ADR(sIPAddr);
	fbGetIPAddr.Len		:= SIZEOF(sIPAddr);
	fbGetIPAddr(enable := FALSE);

	fbGetSubnetMask.pDevice		:= ADR(p_sDevice);
	fbGetSubnetMask.pSubnetMask	:= ADR(sSubnetMask);
	fbGetSubnetMask.Len			:= SIZEOF(sSubnetMask);
	fbGetSubnetMask(enable := FALSE);

	fbGetMacAddr.pDevice	:= ADR(p_sDevice);
	fbGetMacAddr.pMacAddr	:= ADR(a_usiMacAddr);
	fbGetMacAddr.Len		:= SIZEOF(a_usiMacAddr);
	fbGetMacAddr(enable := FALSE);

	fbSetIPAddr.pDevice	:= ADR(p_sDevice);
	fbSetIPAddr.pIPAddr	:= ADR(p_sSetIPAddr);
	fbSetIPAddr.Option	:= cfgOPTION_NON_VOLATILE;
	fbSetIPAddr(enable := FALSE);

	fbSetSubnetMask.pDevice		:= ADR(p_sDevice);
	fbSetSubnetMask.pSubnetMask	:= ADR(p_sSetSubnetMask);
	fbSetSubnetMask.Option		:= cfgOPTION_NON_VOLATILE;
	fbSetSubnetMask(enable := FALSE);

	fbGetETHConfigMode.pDevice	:= ADR(p_sDevice);
	fbGetETHConfigMode(enable := FALSE);

	fbSetETHConfigMode.pDevice		:= ADR(p_sDevice);
	fbSetETHConfigMode.Option		:= cfgOPTION_NON_VOLATILE;
	fbSetETHConfigMode(enable := FALSE);

	fbSetDefaultGateway.pDevice		:= ADR(p_sDevice);
	fbSetDefaultGateway.pGateway	:= ADR(p_sSetDefaultGW);
	fbSetDefaultGateway.Option		:= cfgOPTION_NON_VOLATILE;
	fbSetDefaultGateway(enable := FALSE);
END_ACTION
```
